KUKA KRL program: MyProgram_044().src

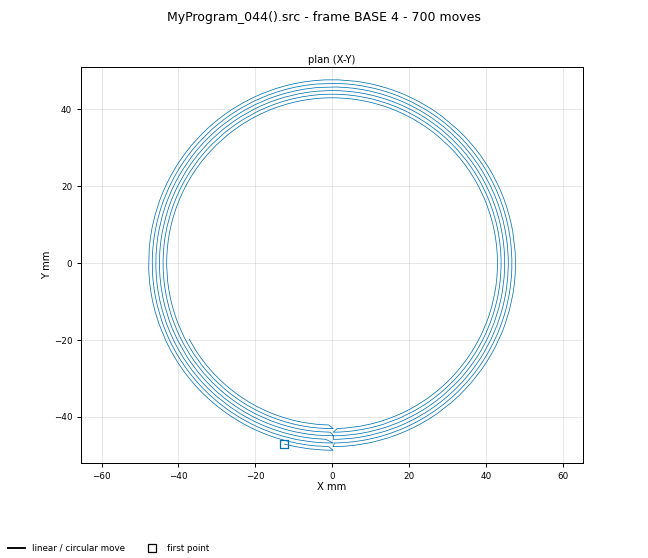
[picture p0: tool path of MyProgram_044().src in frame BASE 4, 700 of 700 moves have a stored position in this frame; points joined in program order, loops and branches not executed]
&ACCESS RVP
&REL 1
&PARAM TEMPLATE = C:\KRC\Roboter\Template\vorgabe
&PARAM EDITMASK = *
DEF MyProgram_044()
; ---- Setting reference (Base) ----
$BASE = BASE_DATA[4]

; --------------------------
; ---- Setting tool (TCP) ----
$TOOL = TOOL_DATA[3]
; --------------------------

$VEL.CP = VEL_APROX_PRINT
Startdeposition()
$VEL.CP = VEL_PRINT
LIN {X -12.395,Y -47.0783,Z 64,A -109.7384,B 24.8767,C -2.5626,E1 24.9625,E2 -526.6882} C_DIS
LIN {X -9.7511,Y -47.6962,Z 64,A -106.6183,B 24.877,C -2.56,E1 24.971,E2 -529.8057} C_DIS
LIN {X -6.2338,Y -48.282,Z 64,A -102.6118,B 24.8774,C -2.5558,E1 24.982,E2 -533.8056} C_DIS
LIN {X -2.3323,Y -48.6268,Z 64,A -98.0603,B 24.8774,C -2.5547,E1 24.9947,E2 -538.3566} C_DIS
LIN {X 0.2772,Y -48.6819,Z 64,A -96.4409,B 24.8798,C -2.5307,E1 24.9991,E2 -539.9189} C_DIS
Enddeposition()
LIN {X 0.2772,Y -48.6819,Z 64,A -96.4409,B 24.8798,C -2.5307,E1 24.9991,E2 -539.9189} C_DIS
Startdeposition()
$VEL.CP = VEL_PRINT
LIN {X -0.9286,Y -47.7351,Z 64,A -98.3994,B 24.879,C -2.5386,E1 24.9937,E2 -537.979} C_DIS
LIN {X -4.5581,Y -47.526,Z 64,A -101.7319,B 24.8774,C -2.5553,E1 24.9845,E2 -534.6849} C_DIS
LIN {X -6.6871,Y -47.2729,Z 64,A -104.8435,B 24.8782,C -2.5471,E1 24.9758,E2 -531.5515} C_DIS
LIN {X -9.333,Y -46.8231,Z 64,A -108.0485,B 24.8781,C -2.5484,E1 24.967,E2 -528.3464} C_DIS
LIN {X -12.0507,Y -46.1979,Z 64,A -111.4661,B 24.8781,C -2.549,E1 24.9577,E2 -524.9256} C_DIS
LIN {X -14.2576,Y -45.5655,Z 64,A -113.9601,B 24.8775,C -2.555,E1 24.9511,E2 -522.4415} C_DIS
LIN {X -16.0969,Y -44.9485,Z 64,A -116.3815,B 24.8775,C -2.5554,E1 24.9447,E2 -520.0165} C_DIS
LIN {X -17.8418,Y -44.2849,Z 64,A -118.4806,B 24.877,C -2.5597,E1 24.9392,E2 -517.923} C_DIS
LIN {X -19.622,Y -43.5255,Z 64,A -120.9789,B 24.877,C -2.5595,E1 24.9328,E2 -515.4183} C_DIS
LIN {X -21.7184,Y -42.5182,Z 64,A -123.9566,B 24.877,C -2.56,E1 24.9254,E2 -512.434} C_DIS
LIN {X -23.6622,Y -41.4683,Z 64,A -126.3379,B 24.8762,C -2.5675,E1 24.9196,E2 -510.0637} C_DIS
LIN {X -25.9488,Y -40.0766,Z 64,A -129.6657,B 24.8759,C -2.5705,E1 24.9117,E2 -506.7327} C_DIS
LIN {X -27.6681,Y -38.9099,Z 64,A -132.1587,B 24.8756,C -2.5746,E1 24.906,E2 -504.2408} C_DIS
LIN {X -29.7267,Y -37.361,Z 64,A -134.9829,B 24.8747,C -2.5838,E1 24.8997,E2 -501.4283} C_DIS
LIN {X -31.3956,Y -35.9696,Z 64,A -138.059,B 24.8748,C -2.5819,E1 24.8932,E2 -498.336} C_DIS
LIN {X -33.6241,Y -33.8958,Z 64,A -141.6218,B 24.874,C -2.5906,E1 24.886,E2 -494.779} C_DIS
LIN {X -35.3679,Y -32.073,Z 64,A -144.7793,B 24.8735,C -2.5952,E1 24.88,E2 -491.6188} C_DIS
LIN {X -37.2668,Y -29.8454,Z 64,A -148.2463,B 24.8727,C -2.6038,E1 24.8738,E2 -488.1564} C_DIS
LIN {X -38.4195,Y -28.3455,Z 64,A -150.8413,B 24.8727,C -2.6048,E1 24.8694,E2 -485.5513} C_DIS
LIN {X -40.21,Y -25.7421,Z 64,A -154.4257,B 24.8714,C -2.6171,E1 24.8639,E2 -481.9782} C_DIS
LIN {X -41.9231,Y -22.8465,Z 64,A -158.8875,B 24.8709,C -2.622,E1 24.8578,E2 -477.5049} C_DIS
LIN {X -43.2781,Y -20.1618,Z 64,A -162.6851,B 24.8702,C -2.6295,E1 24.8532,E2 -473.7045} C_DIS
LIN {X -45.1395,Y -15.5552,Z 64,A -168.6201,B 24.8684,C -2.6469,E1 24.8474,E2 -467.7776} C_DIS
LIN {X -46.1878,Y -12.0906,Z 64,A -172.3555,B 24.8664,C -2.6677,E1 24.8446,E2 -464.0703} C_DIS
LIN {X -46.7423,Y -9.73,Z 64,A -175.6447,B 24.866,C -2.6715,E1 24.8426,E2 -460.771} C_DIS
LIN {X -47.2314,Y -6.9813,Z 64,A -178.6079,B 24.8644,C -2.6868,E1 24.8413,E2 -457.8267} C_DIS
LIN {X -47.4828,Y -4.9862,Z 64,A 178.9355,B 24.8637,C -2.6937,E1 24.8405,E2 -455.3719} C_DIS
LIN {X -47.6696,Y -2.665,Z 64,A 176.3561,B 24.8626,C -2.7052,E1 24.84,E2 -452.8044} C_DIS
LIN {X -47.7273,Y -1.2631,Z 64,A 173.6261,B 24.8634,C -2.6971,E1 24.8398,E2 -450.0386} C_DIS
LIN {X -47.5831,Y 3.9179,Z 64,A 168.1994,B 24.8604,C -2.7268,E1 24.8405,E2 -444.6502} C_DIS
LIN {X -47.2564,Y 6.8067,Z 64,A 164.3377,B 24.8597,C -2.7329,E1 24.8418,E2 -440.7803} C_DIS
LIN {X -46.8079,Y 9.409,Z 64,A 161.4797,B 24.8583,C -2.7468,E1 24.8433,E2 -437.9385} C_DIS
LIN {X -46.0261,Y 12.6919,Z 64,A 156.8291,B 24.8578,C -2.7516,E1 24.8465,E2 -433.2723} C_DIS
LIN {X -44.8495,Y 16.3711,Z 64,A 153.1258,B 24.8551,C -2.7777,E1 24.8497,E2 -429.6103} C_DIS
LIN {X -44.1797,Y 18.1013,Z 64,A 150.357,B 24.8551,C -2.7773,E1 24.8526,E2 -426.8251} C_DIS
LIN {X -43.1295,Y 20.4774,Z 64,A 147.3798,B 24.854,C -2.7883,E1 24.8561,E2 -423.8579} C_DIS
LIN {X -42.0435,Y 22.6245,Z 64,A 143.9498,B 24.8538,C -2.7896,E1 24.8605,E2 -420.4125} C_DIS
LIN {X -40.5413,Y 25.2173,Z 64,A 140.8516,B 24.8521,C -2.8061,E1 24.8649,E2 -417.338} C_DIS
LIN {X -39.3814,Y 26.993,Z 64,A 138.1652,B 24.8515,C -2.8112,E1 24.8691,E2 -414.6502} C_DIS
LIN {X -38.0323,Y 28.8634,Z 64,A 135.3123,B 24.8509,C -2.8173,E1 24.8739,E2 -411.7984} C_DIS
LIN {X -36.3497,Y 30.9548,Z 64,A 132.0941,B 24.85,C -2.8256,E1 24.8796,E2 -408.5849} C_DIS
LIN {X -33.8073,Y 33.7137,Z 64,A 127.1095,B 24.8496,C -2.8299,E1 24.8892,E2 -403.5891} C_DIS
LIN {X -31.9372,Y 35.4898,Z 64,A 124.4061,B 24.8482,C -2.8422,E1 24.8947,E2 -400.9042} C_DIS
LIN {X -29.5152,Y 37.5281,Z 64,A 120.5281,B 24.8475,C -2.8493,E1 24.9031,E2 -397.0284} C_DIS
LIN {X -27.7313,Y 38.8648,Z 64,A 117.8178,B 24.847,C -2.8541,E1 24.9092,E2 -394.3202} C_DIS
LIN {X -25.7301,Y 40.2177,Z 64,A 114.9913,B 24.8463,C -2.8606,E1 24.9158,E2 -391.4999} C_DIS
LIN {X -22.9528,Y 41.8654,Z 64,A 111.0966,B 24.8456,C -2.867,E1 24.9253,E2 -387.609} C_DIS
LIN {X -20.5095,Y 43.1143,Z 64,A 107.8779,B 24.8449,C -2.8732,E1 24.9333,E2 -384.3968} C_DIS
LIN {X -18.1914,Y 44.1428,Z 64,A 104.6647,B 24.8447,C -2.8751,E1 24.9416,E2 -381.1804} C_DIS
LIN {X -14.6042,Y 45.4553,Z 64,A 99.8433,B 24.8445,C -2.8771,E1 24.9543,E2 -376.3547} C_DIS
LIN {X -11.9557,Y 46.2229,Z 64,A 97.1011,B 24.8432,C -2.8889,E1 24.9616,E2 -373.6364} C_DIS
LIN {X -9.839,Y 46.7195,Z 64,A 94.3332,B 24.8432,C -2.8889,E1 24.9692,E2 -370.8646} C_DIS
LIN {X -7.3492,Y 47.1751,Z 64,A 91.1356,B 24.8432,C -2.8885,E1 24.978,E2 -367.6633} C_DIS
LIN {X -4.4968,Y 47.5319,Z 64,A 88.0845,B 24.8424,C -2.8966,E1 24.9864,E2 -364.6294} C_DIS
LIN {X -1.7768,Y 47.7113,Z 64,A 84.2696,B 24.8431,C -2.8893,E1 24.9971,E2 -360.7961} C_DIS
LIN {X 1.6532,Y 47.7156,Z 64,A 79.8522,B 24.8436,C -2.8851,E1 25.0094,E2 -356.3695} C_DIS
LIN {X 5.8821,Y 47.3806,Z 64,A 75.7338,B 24.842,C -2.9002,E1 25.0208,E2 -352.2894} C_DIS
LIN {X 7.6244,Y 47.132,Z 64,A 72.7996,B 24.8435,C -2.8862,E1 25.029,E2 -349.3248} C_DIS
LIN {X 10.1643,Y 46.6496,Z 64,A 70.1964,B 24.8427,C -2.893,E1 25.036,E2 -346.741} C_DIS
LIN {X 12.1272,Y 46.178,Z 64,A 67.8281,B 24.8427,C -2.8925,E1 25.0424,E2 -344.3751} C_DIS
LIN {X 14.1267,Y 45.6062,Z 64,A 65.4726,B 24.8427,C -2.8931,E1 25.0487,E2 -342.025} C_DIS
LIN {X 15.6089,Y 45.1209,Z 64,A 63.3651,B 24.8433,C -2.8876,E1 25.0543,E2 -339.9085} C_DIS
LIN {X 17.816,Y 44.2953,Z 64,A 60.7762,B 24.8432,C -2.889,E1 25.061,E2 -337.3286} C_DIS
LIN {X 19.3175,Y 43.6614,Z 64,A 58.381,B 24.8442,C -2.8794,E1 25.0672,E2 -334.9163} C_DIS
LIN {X 21.7553,Y 42.4995,Z 64,A 55.2848,B 24.8444,C -2.8779,E1 25.075,E2 -331.8251} C_DIS
LIN {X 24.4911,Y 40.9843,Z 64,A 51.7991,B 24.8444,C -2.8774,E1 25.0834,E2 -328.3485} C_DIS
LIN {X 26.3871,Y 39.7898,Z 64,A 48.834,B 24.8454,C -2.8684,E1 25.0904,E2 -325.3718} C_DIS
LIN {X 28.4987,Y 38.3058,Z 64,A 45.1897,B 24.847,C -2.8536,E1 25.0986,E2 -321.7051} C_DIS
LIN {X 32.9673,Y 34.5352,Z 64,A 38.7549,B 24.8473,C -2.8505,E1 25.1121,E2 -315.2885} C_DIS
LIN {X 34.8438,Y 32.6407,Z 64,A 35.5678,B 24.848,C -2.844,E1 25.1183,E2 -312.0996} C_DIS
LIN {X 37.3566,Y 29.7323,Z 64,A 31.3931,B 24.8483,C -2.8416,E1 25.1258,E2 -307.9382} C_DIS
LIN {X 38.7827,Y 27.8463,Z 64,A 27.8779,B 24.8504,C -2.8222,E1 25.1317,E2 -304.3942} C_DIS
LIN {X 40.8107,Y 24.7787,Z 64,A 23.5188,B 24.8515,C -2.812,E1 25.1382,E2 -300.0329} C_DIS
LIN {X 42.0195,Y 22.6688,Z 64,A 20.888,B 24.8517,C -2.8096,E1 25.1417,E2 -297.4101} C_DIS
LIN {X 43.5018,Y 19.6746,Z 64,A 17.248,B 24.8521,C -2.8056,E1 25.1461,E2 -293.7802} C_DIS
LIN {X 44.5986,Y 17.0433,Z 64,A 13.8143,B 24.8532,C -2.7957,E1 25.1497,E2 -290.342} C_DIS
LIN {X 45.4386,Y 14.657,Z 64,A 10.0859,B 24.8555,C -2.7737,E1 25.1531,E2 -286.5826} C_DIS
LIN {X 46.4419,Y 11.0739,Z 64,A 6.0353,B 24.8561,C -2.7683,E1 25.1559,E2 -282.5425} C_DIS
LIN {X 47.015,Y 8.3123,Z 64,A 1.8245,B 24.8588,C -2.7422,E1 25.1581,E2 -278.2946} C_DIS
LIN {X 47.6603,Y 2.8333,Z 64,A -3.3532,B 24.858,C -2.7494,E1 25.1595,E2 -273.1646} C_DIS
LIN {X 47.7412,Y -0.5621,Z 64,A -7.8342,B 24.8602,C -2.7287,E1 25.1597,E2 -268.6614} C_DIS
LIN {X 47.6513,Y -2.9787,Z 64,A -10.826,B 24.8613,C -2.7179,E1 25.1593,E2 -265.6617} C_DIS
LIN {X 47.4135,Y -5.6084,Z 64,A -14.0861,B 24.8625,C -2.7061,E1 25.1584,E2 -262.3931} C_DIS
LIN {X 47.0566,Y -8.0754,Z 64,A -17.2852,B 24.8638,C -2.6928,E1 25.1569,E2 -259.1812} C_DIS
LIN {X 46.1862,Y -12.0964,Z 64,A -22.4469,B 24.8658,C -2.6731,E1 25.1535,E2 -254.003} C_DIS
LIN {X 44.9125,Y -16.1976,Z 64,A -26.7244,B 24.8658,C -2.6742,E1 25.1498,E2 -249.7522} C_DIS
LIN {X 44.2181,Y -18.0066,Z 64,A -29.8233,B 24.8679,C -2.6524,E1 25.1466,E2 -246.6189} C_DIS
LIN {X 42.6286,Y -21.5011,Z 64,A -33.8951,B 24.8682,C -2.6491,E1 25.1417,E2 -242.5612} C_DIS
LIN {X 41.547,Y -23.5236,Z 64,A -36.6489,B 24.869,C -2.6412,E1 25.1379,E2 -239.8031} C_DIS
LIN {X 39.9965,Y -26.0726,Z 64,A -39.9883,B 24.8695,C -2.6359,E1 25.133,E2 -236.4678} C_DIS
LIN {X 38.9178,Y -27.657,Z 64,A -42.8338,B 24.8712,C -2.6194,E1 25.1284,E2 -233.5972} C_DIS
LIN {X 36.2013,Y -31.1289,Z 64,A -48.2812,B 24.8728,C -2.6028,E1 25.1187,E2 -228.1358} C_DIS
LIN {X 33.0813,Y -34.4257,Z 64,A -52.6432,B 24.8721,C -2.61,E1 25.1103,E2 -223.8094} C_DIS
LIN {X 31.1165,Y -36.2119,Z 64,A -56.8723,B 24.8747,C -2.5835,E1 25.1013,E2 -219.5346} C_DIS
LIN {X 27.4183,Y -39.0865,Z 64,A -62.2626,B 24.8754,C -2.5762,E1 25.0893,E2 -214.1462} C_DIS
LIN {X 24.9285,Y -40.7196,Z 64,A -65.4708,B 24.8754,C -2.5762,E1 25.0817,E2 -210.9481} C_DIS
LIN {X 22.8449,Y -41.9239,Z 64,A -68.1053,B 24.8754,C -2.5757,E1 25.0753,E2 -208.3202} C_DIS
LIN {X 21.2981,Y -42.7305,Z 64,A -70.0628,B 24.8755,C -2.5747,E1 25.0705,E2 -206.3658} C_DIS
LIN {X 19.467,Y -43.5948,Z 64,A -72.895,B 24.8766,C -2.5638,E1 25.0632,E2 -203.515} C_DIS
LIN {X 16.541,Y -44.7873,Z 64,A -76.6485,B 24.877,C -2.5594,E1 25.0534,E2 -199.7592} C_DIS
LIN {X 14.4167,Y -45.5152,Z 64,A -79.4404,B 24.8775,C -2.5545,E1 25.046,E2 -196.9609} C_DIS
LIN {X 11.2342,Y -46.4033,Z 64,A -83.1494,B 24.8775,C -2.5548,E1 25.036,E2 -193.2586} C_DIS
LIN {X 9.527,Y -46.7839,Z 64,A -85.5211,B 24.8781,C -2.5484,E1 25.0295,E2 -190.8745} C_DIS
LIN {X 5.9203,Y -47.376,Z 64,A -89.4382,B 24.8776,C -2.5533,E1 25.0187,E2 -186.9727} C_DIS
LIN {X 3.4815,Y -47.6175,Z 64,A -92.9139,B 24.8786,C -2.5429,E1 25.009,E2 -183.4742} C_DIS
LIN {X 0.2827,Y -47.7422,Z 64,A -96.3741,B 24.8781,C -2.548,E1 24.9994,E2 -180.0269} C_DIS
Enddeposition()
LIN {X 0.2827,Y -47.7422,Z 64,A -96.3741,B 24.8781,C -2.548,E1 24.9994,E2 -180.0269} C_DIS
Startdeposition()
$VEL.CP = VEL_PRINT
LIN {X 0.6342,Y -46.8012,Z 64,A -94.7946,B 24.8747,C -2.5833,E1 25.004,E2 -181.6901} C_DIS
LIN {X 3.085,Y -46.7035,Z 64,A -91.5094,B 24.8741,C -2.5892,E1 25.0132,E2 -184.9881} C_DIS
LIN {X 5.746,Y -46.4516,Z 64,A -88.1759,B 24.8739,C -2.5921,E1 25.0225,E2 -188.3263} C_DIS
LIN {X 8.6832,Y -45.9928,Z 64,A -84.6953,B 24.8739,C -2.5921,E1 25.032,E2 -191.8032} C_DIS
LIN {X 11.2628,Y -45.4303,Z 64,A -81.3653,B 24.8734,C -2.5969,E1 25.0411,E2 -195.1398} C_DIS
LIN {X 13.3341,Y -44.8658,Z 64,A -79.1038,B 24.8737,C -2.5933,E1 25.0472,E2 -197.3892} C_DIS
LIN {X 15.2084,Y -44.2657,Z 64,A -76.2089,B 24.8726,C -2.6048,E1 25.0549,E2 -200.3056} C_DIS
LIN {X 17.9227,Y -43.2382,Z 64,A -72.9255,B 24.8726,C -2.6048,E1 25.0634,E2 -203.5819} C_DIS
LIN {X 19.8547,Y -42.3857,Z 64,A -70.4518,B 24.8724,C -2.6068,E1 25.0697,E2 -206.054} C_DIS
LIN {X 21.779,Y -41.4296,Z 64,A -68.1334,B 24.8725,C -2.6055,E1 25.0754,E2 -208.3629} C_DIS
LIN {X 23.3037,Y -40.5916,Z 64,A -65.6769,B 24.8716,C -2.6151,E1 25.0814,E2 -210.8349} C_DIS
LIN {X 24.9354,Y -39.6105,Z 64,A -63.532,B 24.8716,C -2.616,E1 25.0865,E2 -212.9752} C_DIS
LIN {X 27.0041,Y -38.2303,Z 64,A -59.9123,B 24.8699,C -2.6325,E1 25.0949,E2 -216.6217} C_DIS
LIN {X 29.2839,Y -36.5134,Z 64,A -56.5753,B 24.8694,C -2.637,E1 25.1023,E2 -219.9569} C_DIS
LIN {X 31.5484,Y -34.5753,Z 64,A -53.3242,B 24.8694,C -2.6378,E1 25.109,E2 -223.1971} C_DIS
LIN {X 32.9023,Y -33.2893,Z 64,A -50.715,B 24.8682,C -2.6492,E1 25.1143,E2 -225.8224} C_DIS
LIN {X 35.0123,Y -31.0632,Z 64,A -47.2319,B 24.8678,C -2.6534,E1 25.1209,E2 -229.3} C_DIS
LIN {X 36.8334,Y -28.8804,Z 64,A -43.3302,B 24.8661,C -2.6703,E1 25.1278,E2 -233.2238} C_DIS
LIN {X 38.3039,Y -26.8994,Z 64,A -40.9216,B 24.8665,C -2.6668,E1 25.1317,E2 -235.6124} C_DIS
LIN {X 39.2605,Y -25.4833,Z 64,A -38.6906,B 24.8656,C -2.6752,E1 25.1351,E2 -237.8521} C_DIS
LIN {X 40.4459,Y -23.5571,Z 64,A -35.7988,B 24.8646,C -2.6853,E1 25.1393,E2 -240.7531} C_DIS
LIN {X 41.8282,Y -21.0041,Z 64,A -32.3163,B 24.8637,C -2.6942,E1 25.1438,E2 -244.2382} C_DIS
LIN {X 43.0084,Y -18.4673,Z 64,A -28.7338,B 24.8623,C -2.7074,E1 25.1479,E2 -247.8323} C_DIS
LIN {X 43.9827,Y -16.0083,Z 64,A -25.6523,B 24.8617,C -2.7141,E1 25.1509,E2 -250.9126} C_DIS
LIN {X 44.7903,Y -13.5846,Z 64,A -22.3402,B 24.8603,C -2.7273,E1 25.1537,E2 -254.2371} C_DIS
LIN {X 45.413,Y -11.3318,Z 64,A -19.2917,B 24.859,C -2.7398,E1 25.1558,E2 -257.2976} C_DIS
LIN {X 46.0028,Y -8.6308,Z 64,A -16.6613,B 24.8594,C -2.7357,E1 25.1573,E2 -259.903} C_DIS
LIN {X 46.339,Y -6.59,Z 64,A -13.4915,B 24.8573,C -2.756,E1 25.1586,E2 -263.1023} C_DIS
LIN {X 46.6589,Y -3.7003,Z 64,A -10.2295,B 24.8568,C -2.7615,E1 25.1595,E2 -266.3577} C_DIS
LIN {X 46.7751,Y -1.6919,Z 64,A -7.9435,B 24.8563,C -2.7658,E1 25.1597,E2 -268.6403} C_DIS
LIN {X 46.7921,Y 1.1,Z 64,A -4.3105,B 24.8548,C -2.7807,E1 25.1597,E2 -272.2869} C_DIS
LIN {X 46.6119,Y 4.247,Z 64,A -0.573,B 24.8537,C -2.7904,E1 25.1589,E2 -276.0252} C_DIS
LIN {X 46.3482,Y 6.5248,Z 64,A 2.0753,B 24.8532,C -2.796,E1 25.1579,E2 -278.6711} C_DIS
LIN {X 46.0174,Y 8.5543,Z 64,A 4.5784,B 24.8524,C -2.8034,E1 25.1567,E2 -281.1771} C_DIS
LIN {X 45.5613,Y 10.7204,Z 64,A 7.2402,B 24.8516,C -2.8106,E1 25.1551,E2 -283.8406} C_DIS
LIN {X 45.1148,Y 12.4653,Z 64,A 9.2143,B 24.8514,C -2.8128,E1 25.1537,E2 -285.8085} C_DIS
LIN {X 44.5439,Y 14.3732,Z 64,A 11.9778,B 24.8499,C -2.8262,E1 25.1514,E2 -288.588} C_DIS
LIN {X 43.6644,Y 16.8579,Z 64,A 15.1569,B 24.8491,C -2.8345,E1 25.1483,E2 -291.769} C_DIS
LIN {X 42.7002,Y 19.1685,Z 64,A 18.2894,B 24.848,C -2.8444,E1 25.1448,E2 -294.9077} C_DIS
LIN {X 41.3826,Y 21.8684,Z 64,A 21.5209,B 24.8478,C -2.846,E1 25.1408,E2 -298.1258} C_DIS
LIN {X 40.1234,Y 24.102,Z 64,A 25.3236,B 24.8456,C -2.8666,E1 25.1354,E2 -301.9577} C_DIS
LIN {X 38.9075,Y 26.0191,Z 64,A 27.9514,B 24.8452,C -2.8708,E1 25.1314,E2 -304.5823} C_DIS
LIN {X 37.0697,Y 28.5758,Z 64,A 31.3241,B 24.8452,C -2.8711,E1 25.1258,E2 -307.9396} C_DIS
LIN {X 34.9763,Y 31.1035,Z 64,A 35.5365,B 24.8438,C -2.8837,E1 25.1182,E2 -312.1627} C_DIS
LIN {X 33.2605,Y 32.9315,Z 64,A 38.6668,B 24.8429,C -2.8914,E1 25.1121,E2 -315.2976} C_DIS
LIN {X 30.5308,Y 35.4771,Z 64,A 43.0808,B 24.8422,C -2.8975,E1 25.103,E2 -319.7084} C_DIS
LIN {X 28.9107,Y 36.8094,Z 64,A 45.5609,B 24.8419,C -2.9006,E1 25.0976,E2 -322.1865} C_DIS
LIN {X 27.5077,Y 37.8695,Z 64,A 47.646,B 24.8416,C -2.9031,E1 25.0929,E2 -324.2699} C_DIS
LIN {X 25.2892,Y 39.3853,Z 64,A 51.0253,B 24.8409,C -2.9099,E1 25.085,E2 -327.6541} C_DIS
LIN {X 23.7995,Y 40.3029,Z 64,A 53.5315,B 24.8399,C -2.9193,E1 25.079,E2 -330.175} C_DIS
LIN {X 20.5147,Y 42.0701,Z 64,A 58.282,B 24.8389,C -2.9283,E1 25.0672,E2 -334.9336} C_DIS
LIN {X 17.0842,Y 43.5761,Z 64,A 62.1836,B 24.8396,C -2.9213,E1 25.0572,E2 -338.8095} C_DIS
LIN {X 15.4042,Y 44.198,Z 64,A 64.4907,B 24.8392,C -2.9251,E1 25.0511,E2 -341.121} C_DIS
LIN {X 13.3641,Y 44.8567,Z 64,A 67.1244,B 24.839,C -2.9272,E1 25.0441,E2 -343.755} C_DIS
LIN {X 10.9256,Y 45.5122,Z 64,A 70.2327,B 24.8388,C -2.9293,E1 25.0357,E2 -346.8635} C_DIS
LIN {X 7.819,Y 46.1476,Z 64,A 73.9653,B 24.8388,C -2.9285,E1 25.0255,E2 -350.5896} C_DIS
LIN {X 5.9098,Y 46.4308,Z 64,A 76.3697,B 24.8388,C -2.9297,E1 25.0188,E2 -352.9949} C_DIS
LIN {X 3.7771,Y 46.6527,Z 64,A 79.2175,B 24.8383,C -2.9335,E1 25.0109,E2 -355.8502} C_DIS
LIN {X 1.1995,Y 46.7899,Z 64,A 83.0787,B 24.8371,C -2.9445,E1 25,E2 -359.7366} C_DIS
LIN {X -3.9742,Y 46.6363,Z 64,A 88.5906,B 24.8388,C -2.9292,E1 24.9848,E2 -365.2136} C_DIS
LIN {X -6.8684,Y 46.2987,Z 64,A 92.4777,B 24.8385,C -2.932,E1 24.974,E2 -369.1102} C_DIS
LIN {X -9.36,Y 45.8599,Z 64,A 95.1805,B 24.8394,C -2.9236,E1 24.9666,E2 -371.7959} C_DIS
LIN {X -11.4862,Y 45.3743,Z 64,A 97.9922,B 24.8394,C -2.9233,E1 24.959,E2 -374.6107} C_DIS
LIN {X -14.1559,Y 44.6132,Z 64,A 101.7915,B 24.8392,C -2.9256,E1 24.9488,E2 -378.4219} C_DIS
LIN {X -16.5969,Y 43.764,Z 64,A 105.3784,B 24.8389,C -2.9278,E1 24.9394,E2 -382.0215} C_DIS
LIN {X -20.1209,Y 42.2596,Z 64,A 109.38,B 24.8408,C -2.9108,E1 24.9293,E2 -385.9923} C_DIS
LIN {X -23.5707,Y 40.4364,Z 64,A 114.4699,B 24.8412,C -2.9073,E1 24.9168,E2 -391.0884} C_DIS
LIN {X -25.9496,Y 38.9535,Z 64,A 117.5019,B 24.8425,C -2.8952,E1 24.9097,E2 -394.1014} C_DIS
LIN {X -27.9755,Y 37.5252,Z 64,A 120.6772,B 24.8429,C -2.8911,E1 24.9026,E2 -397.278} C_DIS
LIN {X -30.2011,Y 35.7586,Z 64,A 124.1179,B 24.8438,C -2.8832,E1 24.8951,E2 -400.7127} C_DIS
LIN {X -31.6166,Y 34.5128,Z 64,A 126.9902,B 24.8435,C -2.8857,E1 24.8892,E2 -403.6028} C_DIS
LIN {X -34.6929,Y 31.4191,Z 64,A 131.8617,B 24.8456,C -2.8665,E1 24.8798,E2 -408.4493} C_DIS
LIN {X -36.4484,Y 29.3645,Z 64,A 135.1345,B 24.8466,C -2.8576,E1 24.874,E2 -411.7159} C_DIS
LIN {X -37.6336,Y 27.8299,Z 64,A 137.8335,B 24.8468,C -2.8557,E1 24.8695,E2 -414.4234} C_DIS
LIN {X -39.4095,Y 25.2514,Z 64,A 141.4179,B 24.8483,C -2.842,E1 24.864,E2 -417.9929} C_DIS
LIN {X -41.0331,Y 22.5172,Z 64,A 145.9162,B 24.8486,C -2.839,E1 24.8577,E2 -422.5076} C_DIS
LIN {X -42.3743,Y 19.8791,Z 64,A 149.375,B 24.8499,C -2.8262,E1 24.8536,E2 -425.9547} C_DIS
LIN {X -43.7887,Y 16.5316,Z 64,A 153.3349,B 24.852,C -2.8066,E1 24.8495,E2 -429.8896} C_DIS
LIN {X -44.6099,Y 14.1663,Z 64,A 156.814,B 24.8524,C -2.8027,E1 24.8464,E2 -433.3792} C_DIS
LIN {X -45.5232,Y 10.8797,Z 64,A 160.7905,B 24.8541,C -2.7872,E1 24.8436,E2 -437.3419} C_DIS
LIN {X -46.0725,Y 8.2504,Z 64,A 163.9661,B 24.8553,C -2.7755,E1 24.842,E2 -440.5082} C_DIS
LIN {X -46.4192,Y 5.9983,Z 64,A 166.8986,B 24.856,C -2.7686,E1 24.8408,E2 -443.4418} C_DIS
LIN {X -46.6752,Y 3.4923,Z 64,A 169.4985,B 24.8577,C -2.7527,E1 24.8402,E2 -446.0192} C_DIS
LIN {X -46.7964,Y 0.9112,Z 64,A 173.5745,B 24.8575,C -2.7545,E1 24.8398,E2 -450.1241} C_DIS
LIN {X -46.7535,Y -2.1957,Z 64,A 176.9979,B 24.8592,C -2.7377,E1 24.8401,E2 -453.5279} C_DIS
LIN {X -46.6217,Y -4.1413,Z 64,A 179.4719,B 24.8599,C -2.7314,E1 24.8407,E2 -456.0016} C_DIS
LIN {X -46.3019,Y -6.85,Z 64,A -177.6073,B 24.8615,C -2.7157,E1 24.8417,E2 -458.9023} C_DIS
LIN {X -46.0802,Y -8.2066,Z 64,A -175.3508,B 24.8613,C -2.718,E1 24.8428,E2 -461.1778} C_DIS
LIN {X -45.4603,Y -11.1404,Z 64,A -171.8246,B 24.8626,C -2.705,E1 24.845,E2 -464.6937} C_DIS
LIN {X -44.2097,Y -15.3707,Z 64,A -166.0866,B 24.8637,C -2.6937,E1 24.8498,E2 -470.4374} C_DIS
LIN {X -43.0201,Y -18.4394,Z 64,A -162.6722,B 24.8657,C -2.6741,E1 24.8533,E2 -473.8241} C_DIS
LIN {X -42.3744,Y -19.8785,Z 64,A -160.6968,B 24.8662,C -2.6694,E1 24.8556,E2 -475.799} C_DIS
LIN {X -41.701,Y -21.2545,Z 64,A -158.4981,B 24.8662,C -2.6686,E1 24.8584,E2 -478.0078} C_DIS
LIN {X -40.4073,Y -23.6221,Z 64,A -155.4706,B 24.8675,C -2.6562,E1 24.8625,E2 -481.0215} C_DIS
LIN {X -39.1654,Y -25.6288,Z 64,A -152.5662,B 24.8682,C -2.6491,E1 24.8669,E2 -483.9237} C_DIS
LIN {X -37.4149,Y -28.1223,Z 64,A -148.5392,B 24.8687,C -2.6442,E1 24.8734,E2 -487.9584} C_DIS
LIN {X -35.6448,Y -30.3346,Z 64,A -144.7853,B 24.8691,C -2.6402,E1 24.8801,E2 -491.7203} C_DIS
LIN {X -33.9869,Y -32.1817,Z 64,A -141.5829,B 24.8695,C -2.636,E1 24.8863,E2 -494.9267} C_DIS
LIN {X -31.8502,Y -34.2976,Z 64,A -138.2021,B 24.8707,C -2.6244,E1 24.8931,E2 -498.2936} C_DIS
LIN {X -29.4531,Y -36.3766,Z 64,A -134.8763,B 24.8722,C -2.6092,E1 24.9001,E2 -501.596} C_DIS
LIN {X -27.4013,Y -37.9465,Z 64,A -131.5451,B 24.8725,C -2.6062,E1 24.9075,E2 -504.932} C_DIS
LIN {X -26.2155,Y -38.7749,Z 64,A -129.4028,B 24.8722,C -2.6088,E1 24.9125,E2 -507.0877} C_DIS
LIN {X -23.7348,Y -40.3412,Z 64,A -125.8842,B 24.8728,C -2.6025,E1 24.9209,E2 -510.6023} C_DIS
LIN {X -21.2142,Y -41.7215,Z 64,A -122.2182,B 24.8731,C -2.6003,E1 24.9299,E2 -514.2731} C_DIS
LIN {X -19.144,Y -42.7112,Z 64,A -119.7825,B 24.8739,C -2.5915,E1 24.9361,E2 -516.694} C_DIS
LIN {X -17.3939,Y -43.4531,Z 64,A -117.2986,B 24.8739,C -2.5916,E1 24.9425,E2 -519.1837} C_DIS
LIN {X -15.3149,Y -44.2293,Z 64,A -114.1502,B 24.8735,C -2.596,E1 24.9508,E2 -522.3487} C_DIS
LIN {X -12.8555,Y -45.0054,Z 64,A -110.7564,B 24.8733,C -2.5976,E1 24.96,E2 -525.752} C_DIS
LIN {X -9.964,Y -45.7325,Z 64,A -107.9206,B 24.8747,C -2.5829,E1 24.9676,E2 -528.5566} C_DIS
LIN {X -8.5188,Y -46.0242,Z 64,A -105.5194,B 24.8739,C -2.5918,E1 24.9742,E2 -530.9814} C_DIS
LIN {X -4.7848,Y -46.56,Z 64,A -101.1924,B 24.8744,C -2.5863,E1 24.9862,E2 -535.2985} C_DIS
LIN {X -2.7262,Y -46.7258,Z 64,A -98.6042,B 24.8744,C -2.5874,E1 24.9934,E2 -537.89} C_DIS
LIN {X 0.2899,Y -46.7986,Z 64,A -96.5083,B 24.8768,C -2.5621,E1 24.9991,E2 -539.9261} C_DIS
Enddeposition()
LIN {X 0.2899,Y -46.7986,Z 64,A -96.5083,B 24.8768,C -2.5621,E1 24.9991,E2 -539.9261} C_DIS
Startdeposition()
$VEL.CP = VEL_PRINT
LIN {X -1.6444,Y -45.8371,Z 64,A -99.7182,B 24.8764,C -2.5659,E1 24.9902,E2 -536.7246} C_DIS
LIN {X -4.8851,Y -45.6056,Z 64,A -102.718,B 24.8748,C -2.5824,E1 24.9819,E2 -533.7626} C_DIS
LIN {X -6.7079,Y -45.3739,Z 64,A -105.1635,B 24.875,C -2.5805,E1 24.9751,E2 -531.3108} C_DIS
LIN {X -8.719,Y -45.0303,Z 64,A -107.7698,B 24.875,C -2.5805,E1 24.968,E2 -528.7018} C_DIS
LIN {X -10.9386,Y -44.5432,Z 64,A -110.5241,B 24.8747,C -2.5831,E1 24.9605,E2 -525.9501} C_DIS
LIN {X -12.6995,Y -44.0734,Z 64,A -113.0005,B 24.8749,C -2.5816,E1 24.9538,E2 -523.4662} C_DIS
LIN {X -15.3679,Y -43.2154,Z 64,A -116.7534,B 24.8749,C -2.5807,E1 24.9439,E2 -519.7041} C_DIS
LIN {X -18.1645,Y -42.1169,Z 64,A -120.156,B 24.8741,C -2.5895,E1 24.9351,E2 -516.3147} C_DIS
LIN {X -20.1395,Y -41.2086,Z 64,A -122.8725,B 24.8738,C -2.5925,E1 24.9282,E2 -513.5986} C_DIS
LIN {X -22.472,Y -39.9847,Z 64,A -125.8961,B 24.873,C -2.6006,E1 24.9208,E2 -510.5857} C_DIS
LIN {X -23.9885,Y -39.0937,Z 64,A -128.8256,B 24.8737,C -2.5935,E1 24.9138,E2 -507.6302} C_DIS
LIN {X -26.2953,Y -37.5804,Z 64,A -132.7571,B 24.8738,C -2.5923,E1 24.9047,E2 -503.6827} C_DIS
LIN {X -29.8183,Y -34.8515,Z 64,A -137.3802,B 24.8716,C -2.6151,E1 24.8947,E2 -499.0966} C_DIS
LIN {X -31.8833,Y -32.9728,Z 64,A -140.9945,B 24.8711,C -2.6203,E1 24.8874,E2 -495.48} C_DIS
LIN {X -33.6222,Y -31.1985,Z 64,A -143.9678,B 24.8703,C -2.6286,E1 24.8816,E2 -492.5136} C_DIS
LIN {X -34.6856,Y -30.0115,Z 64,A -146.5806,B 24.8706,C -2.6248,E1 24.8768,E2 -489.88} C_DIS
LIN {X -36.5496,Y -27.7114,Z 64,A -150.6684,B 24.8703,C -2.6285,E1 24.8698,E2 -485.7815} C_DIS
LIN {X -38.5002,Y -24.9302,Z 64,A -154.9483,B 24.8693,C -2.6387,E1 24.8632,E2 -481.5045} C_DIS
LIN {X -40.1793,Y -22.1229,Z 64,A -157.9202,B 24.8668,C -2.6634,E1 24.8592,E2 -478.5763} C_DIS
LIN {X -41.1239,Y -20.3117,Z 64,A -160.8046,B 24.8665,C -2.6661,E1 24.8555,E2 -475.6829} C_DIS
LIN {X -42.2059,Y -17.956,Z 64,A -164.2136,B 24.8658,C -2.673,E1 24.8516,E2 -472.2715} C_DIS
LIN {X -43.2718,Y -15.2087,Z 64,A -168.0594,B 24.865,C -2.6815,E1 24.8479,E2 -468.4244} C_DIS
LIN {X -44.301,Y -11.8818,Z 64,A -171.9257,B 24.8631,C -2.7003,E1 24.8449,E2 -464.5807} C_DIS
LIN {X -44.8135,Y -9.7725,Z 64,A -174.9708,B 24.8627,C -2.7044,E1 24.843,E2 -461.5274} C_DIS
LIN {X -45.2438,Y -7.533,Z 64,A -177.4649,B 24.8613,C -2.7174,E1 24.8418,E2 -459.0498} C_DIS
LIN {X -45.5066,Y -5.7371,Z 64,A -179.9593,B 24.8609,C -2.7216,E1 24.8408,E2 -456.5505} C_DIS
LIN {X -45.7487,Y -3.2846,Z 64,A 176.8311,B 24.8601,C -2.7296,E1 24.84,E2 -453.3407} C_DIS
LIN {X -45.8575,Y -0.9171,Z 64,A 173.6759,B 24.8594,C -2.7365,E1 24.8398,E2 -450.1829} C_DIS
LIN {X -45.8059,Y 2.3515,Z 64,A 169.7422,B 24.8578,C -2.7511,E1 24.8401,E2 -446.2606} C_DIS
LIN {X -45.6107,Y 4.8396,Z 64,A 166.6976,B 24.8567,C -2.7618,E1 24.8409,E2 -443.2232} C_DIS
LIN {X -45.3173,Y 7.0778,Z 64,A 163.9254,B 24.8558,C -2.7712,E1 24.842,E2 -440.4571} C_DIS
LIN {X -45.047,Y 8.6319,Z 64,A 161.476,B 24.8558,C -2.7715,E1 24.8433,E2 -437.994} C_DIS
LIN {X -44.2224,Y 12.1705,Z 64,A 157.0419,B 24.8541,C -2.7868,E1 24.8463,E2 -433.5706} C_DIS
LIN {X -43.4522,Y 14.6849,Z 64,A 154.1452,B 24.8526,C -2.8016,E1 24.8487,E2 -430.6926} C_DIS
LIN {X -42.8802,Y 16.28,Z 64,A 151.7301,B 24.8523,C -2.8043,E1 24.8511,E2 -428.2704} C_DIS
LIN {X -41.8108,Y 18.8572,Z 64,A 148.2049,B 24.8512,C -2.8141,E1 24.855,E2 -424.7492} C_DIS
LIN {X -40.7314,Y 21.0881,Z 64,A 145.3361,B 24.85,C -2.8259,E1 24.8585,E2 -421.8931} C_DIS
LIN {X -39.766,Y 22.8564,Z 64,A 142.6406,B 24.8495,C -2.8308,E1 24.8622,E2 -419.1952} C_DIS
LIN {X -38.8342,Y 24.4063,Z 64,A 139.9723,B 24.8493,C -2.832,E1 24.8662,E2 -416.5161} C_DIS
LIN {X -36.6076,Y 27.6342,Z 64,A 135.6592,B 24.8471,C -2.8524,E1 24.8731,E2 -412.2307} C_DIS
LIN {X -35.2612,Y 29.3325,Z 64,A 132.5107,B 24.8471,C -2.8537,E1 24.8787,E2 -409.0707} C_DIS
LIN {X -33.5949,Y 31.2278,Z 64,A 129.363,B 24.8462,C -2.8615,E1 24.8846,E2 -405.9276} C_DIS
LIN {X -31.486,Y 33.3525,Z 64,A 125.9701,B 24.8447,C -2.8747,E1 24.8913,E2 -402.5521} C_DIS
LIN {X -29.948,Y 34.7405,Z 64,A 123.6132,B 24.8438,C -2.8835,E1 24.8962,E2 -400.2068} C_DIS
LIN {X -28.5423,Y 35.9041,Z 64,A 120.9883,B 24.8438,C -2.8838,E1 24.9019,E2 -397.5728} C_DIS
LIN {X -25.5389,Y 38.0989,Z 64,A 116.302,B 24.8428,C -2.8925,E1 24.9126,E2 -392.8909} C_DIS
LIN {X -22.8772,Y 39.754,Z 64,A 111.7336,B 24.843,C -2.8907,E1 24.9235,E2 -388.3044} C_DIS
LIN {X -19.9461,Y 41.3026,Z 64,A 107.6538,B 24.8422,C -2.898,E1 24.9337,E2 -384.2313} C_DIS
LIN {X -16.4279,Y 42.8239,Z 64,A 103.6415,B 24.8403,C -2.9154,E1 24.944,E2 -380.2513} C_DIS
LIN {X -15.1283,Y 43.2998,Z 64,A 101.428,B 24.8408,C -2.9107,E1 24.9498,E2 -378.0223} C_DIS
LIN {X -12.4332,Y 44.1494,Z 64,A 97.9036,B 24.8404,C -2.9146,E1 24.9593,E2 -374.5012} C_DIS
LIN {X -9.4352,Y 44.8855,Z 64,A 94.2735,B 24.8396,C -2.9213,E1 24.9691,E2 -370.8823} C_DIS
LIN {X -7.2288,Y 45.294,Z 64,A 91.431,B 24.8395,C -2.9228,E1 24.9769,E2 -368.0405} C_DIS
LIN {X -4.7444,Y 45.6206,Z 64,A 88.5263,B 24.8389,C -2.9279,E1 24.985,E2 -365.146} C_DIS
LIN {X -3.2274,Y 45.7526,Z 64,A 85.7364,B 24.8403,C -2.9155,E1 24.9928,E2 -362.3257} C_DIS
LIN {X 1.0048,Y 45.8558,Z 64,A 81.1245,B 24.839,C -2.9268,E1 25.0056,E2 -357.7406} C_DIS
LIN {X 3.3168,Y 45.747,Z 64,A 78.3493,B 24.8388,C -2.9286,E1 25.0133,E2 -354.9707} C_DIS
LIN {X 5.485,Y 45.5376,Z 64,A 75.4286,B 24.8392,C -2.9251,E1 25.0215,E2 -352.0438} C_DIS
LIN {X 8.0141,Y 45.1611,Z 64,A 72.4582,B 24.8389,C -2.9277,E1 25.0296,E2 -349.0823} C_DIS
LIN {X 9.6602,Y 44.838,Z 64,A 70.0781,B 24.8395,C -2.9222,E1 25.0362,E2 -346.6923} C_DIS
LIN {X 12.4449,Y 44.1461,Z 64,A 66.3288,B 24.8401,C -2.9174,E1 25.0463,E2 -342.9374} C_DIS
LIN {X 15.1996,Y 43.275,Z 64,A 62.9616,B 24.84,C -2.9184,E1 25.0552,E2 -339.579} C_DIS
LIN {X 17.5757,Y 42.3659,Z 64,A 59.7085,B 24.8404,C -2.9141,E1 25.0636,E2 -336.3229} C_DIS
LIN {X 19.8447,Y 41.3514,Z 64,A 56.7665,B 24.8405,C -2.9132,E1 25.0711,E2 -333.3864} C_DIS
LIN {X 21.9899,Y 40.2518,Z 64,A 53.6678,B 24.8411,C -2.9079,E1 25.0787,E2 -330.2837} C_DIS
LIN {X 24.1788,Y 38.9762,Z 64,A 50.7667,B 24.8411,C -2.9077,E1 25.0857,E2 -327.3913} C_DIS
LIN {X 26.1545,Y 37.6788,Z 64,A 47.714,B 24.8418,C -2.9014,E1 25.0928,E2 -324.3337} C_DIS
LIN {X 27.8331,Y 36.4566,Z 64,A 45.2832,B 24.842,C -2.8997,E1 25.0982,E2 -321.9077} C_DIS
LIN {X 28.9991,Y 35.5363,Z 64,A 43.1912,B 24.8428,C -2.8923,E1 25.1028,E2 -319.8059} C_DIS
LIN {X 30.8372,Y 33.9534,Z 64,A 40.2316,B 24.8433,C -2.8877,E1 25.109,E2 -316.8471} C_DIS
LIN {X 32.5275,Y 32.3378,Z 64,A 36.5786,B 24.8454,C -2.8689,E1 25.1163,E2 -313.1651} C_DIS
LIN {X 34.5974,Y 30.1127,Z 64,A 33.1844,B 24.8455,C -2.8675,E1 25.1225,E2 -309.7828} C_DIS
LIN {X 36.3961,Y 27.912,Z 64,A 29.8786,B 24.8459,C -2.8636,E1 25.1283,E2 -306.4831} C_DIS
LIN {X 37.9853,Y 25.7074,Z 64,A 26.786,B 24.8463,C -2.8607,E1 25.1332,E2 -303.3988} C_DIS
LIN {X 39.374,Y 23.5257,Z 64,A 22.9388,B 24.8483,C -2.8413,E1 25.1389,E2 -299.5252} C_DIS
LIN {X 41.2674,Y 20.018,Z 64,A 18.1107,B 24.8495,C -2.8306,E1 25.1451,E2 -294.6975} C_DIS
LIN {X 42.3522,Y 17.6085,Z 64,A 15.2349,B 24.8496,C -2.8291,E1 25.1482,E2 -291.8338} C_DIS
LIN {X 43.065,Y 15.785,Z 64,A 12.8325,B 24.8503,C -2.8229,E1 25.1506,E2 -289.4301} C_DIS
LIN {X 43.6393,Y 14.1196,Z 64,A 10.753,B 24.8507,C -2.8187,E1 25.1525,E2 -287.3524} C_DIS
LIN {X 44.4922,Y 11.1453,Z 64,A 5.9316,B 24.8538,C -2.7897,E1 25.156,E2 -282.49} C_DIS
LIN {X 45.1439,Y 8.1102,Z 64,A 2.7608,B 24.8537,C -2.7909,E1 25.1576,E2 -279.3406} C_DIS
LIN {X 45.6093,Y 4.8505,Z 64,A -1.8445,B 24.856,C -2.7691,E1 25.1592,E2 -274.7109} C_DIS
LIN {X 45.8417,Y 1.5115,Z 64,A -5.3017,B 24.856,C -2.7695,E1 25.1597,E2 -271.2751} C_DIS
LIN {X 45.8648,Y -0.467,Z 64,A -8.4837,B 24.8581,C -2.7485,E1 25.1597,E2 -268.0624} C_DIS
LIN {X 45.7069,Y -3.8277,Z 64,A -12.7728,B 24.8596,C -2.7337,E1 25.1588,E2 -263.7638} C_DIS
LIN {X 45.3349,Y -6.964,Z 64,A -15.6802,B 24.8589,C -2.7406,E1 25.1577,E2 -260.8898} C_DIS
LIN {X 44.9583,Y -9.0839,Z 64,A -18.7975,B 24.8606,C -2.7242,E1 25.1561,E2 -257.752} C_DIS
LIN {X 44.488,Y -11.1621,Z 64,A -20.9937,B 24.8606,C -2.7246,E1 25.1547,E2 -255.5695} C_DIS
LIN {X 43.8702,Y -13.3845,Z 64,A -24.4299,B 24.8625,C -2.7054,E1 25.152,E2 -252.1075} C_DIS
LIN {X 42.9193,Y -16.1767,Z 64,A -28.2089,B 24.8639,C -2.6925,E1 25.1484,E2 -248.3192} C_DIS
LIN {X 41.4028,Y -19.7368,Z 64,A -32.3715,B 24.864,C -2.6906,E1 25.1437,E2 -244.1747} C_DIS
LIN {X 39.575,Y -23.1861,Z 64,A -36.9697,B 24.8649,C -2.6818,E1 25.1376,E2 -239.5798} C_DIS
LIN {X 38.6817,Y -24.6472,Z 64,A -39.5224,B 24.8663,C -2.6682,E1 25.1338,E2 -237.0079} C_DIS
LIN {X 37.4756,Y -26.4456,Z 64,A -42.1492,B 24.8669,C -2.6623,E1 25.1297,E2 -234.38} C_DIS
LIN {X 35.9802,Y -28.446,Z 64,A -45.5525,B 24.8682,C -2.6489,E1 25.1239,E2 -230.9612} C_DIS
LIN {X 34.4969,Y -30.2278,Z 64,A -48.0233,B 24.8682,C -2.6493,E1 25.1194,E2 -228.5025} C_DIS
LIN {X 33.3098,Y -31.5313,Z 64,A -50.2294,B 24.8688,C -2.6438,E1 25.1152,E2 -226.2931} C_DIS
LIN {X 31.5735,Y -33.2702,Z 64,A -53.7566,B 24.8703,C -2.6284,E1 25.1081,E2 -222.7441} C_DIS
LIN {X 29.7687,Y -34.8938,Z 64,A -56.2806,B 24.8701,C -2.6306,E1 25.1028,E2 -220.2354} C_DIS
LIN {X 28.4198,Y -36.0009,Z 64,A -58.4133,B 24.8704,C -2.6268,E1 25.0982,E2 -218.1017} C_DIS
LIN {X 26.5914,Y -37.3718,Z 64,A -61.6578,B 24.8717,C -2.6141,E1 25.0909,E2 -214.8387} C_DIS
LIN {X 24.5847,Y -38.7213,Z 64,A -64.5152,B 24.872,C -2.6112,E1 25.0842,E2 -211.9838} C_DIS
LIN {X 21.8554,Y -40.3248,Z 64,A -68.5319,B 24.8728,C -2.6032,E1 25.0744,E2 -207.9601} C_DIS
LIN {X 19.0481,Y -41.7244,Z 64,A -72.4987,B 24.8735,C -2.5962,E1 25.0644,E2 -203.9871} C_DIS
LIN {X 16.9466,Y -42.6211,Z 64,A -76.3558,B 24.8755,C -2.5755,E1 25.0543,E2 -200.0895} C_DIS
LIN {X 13.774,Y -43.7495,Z 64,A -80.0599,B 24.8752,C -2.5788,E1 25.0445,E2 -196.4002} C_DIS
LIN {X 9.7338,Y -44.8219,Z 64,A -84.4549,B 24.8743,C -2.5873,E1 25.0327,E2 -192.0319} C_DIS
LIN {X 7.8299,Y -45.193,Z 64,A -87.0031,B 24.8747,C -2.5833,E1 25.0257,E2 -189.4771} C_DIS
LIN {X 5.5797,Y -45.5262,Z 64,A -90.2535,B 24.8755,C -2.5749,E1 25.0166,E2 -186.2094} C_DIS
LIN {X 1.7385,Y -45.8341,Z 64,A -94.3572,B 24.8746,C -2.5842,E1 25.0052,E2 -182.1294} C_DIS
LIN {X 0.2949,Y -45.8474,Z 64,A -96.4193,B 24.875,C -2.5799,E1 24.9995,E2 -180.0574} C_DIS
Enddeposition()
LIN {X 0.2949,Y -45.8474,Z 64,A -96.4193,B 24.875,C -2.5799,E1 24.9995,E2 -180.0574} C_DIS
Startdeposition()
$VEL.CP = VEL_PRINT
LIN {X 0.3744,Y -44.9265,Z 64,A -94.9095,B 24.8713,C -2.6181,E1 25.0039,E2 -181.6579} C_DIS
LIN {X 2.7497,Y -44.8434,Z 64,A -91.839,B 24.8711,C -2.6199,E1 25.0125,E2 -184.7316} C_DIS
LIN {X 5.4133,Y -44.6009,Z 64,A -88.7779,B 24.8715,C -2.6161,E1 25.021,E2 -187.7817} C_DIS
LIN {X 6.9676,Y -44.3845,Z 64,A -86.4066,B 24.8708,C -2.6235,E1 25.0276,E2 -190.1685} C_DIS
LIN {X 9.5676,Y -43.8974,Z 64,A -82.9038,B 24.8703,C -2.6285,E1 25.0372,E2 -193.6788} C_DIS
LIN {X 12.9001,Y -43.0359,Z 64,A -79.0674,B 24.8707,C -2.6239,E1 25.0475,E2 -197.4981} C_DIS
LIN {X 14.6528,Y -42.4716,Z 64,A -76.5523,B 24.8702,C -2.6296,E1 25.0541,E2 -200.0217} C_DIS
LIN {X 17.3456,Y -41.4447,Z 64,A -72.8944,B 24.8697,C -2.6343,E1 25.0636,E2 -203.6826} C_DIS
LIN {X 19.1164,Y -40.6583,Z 64,A -70.2847,B 24.8691,C -2.6404,E1 25.0703,E2 -206.3003} C_DIS
LIN {X 21.675,Y -39.3543,Z 64,A -66.5433,B 24.8683,C -2.6479,E1 25.0795,E2 -210.0489} C_DIS
LIN {X 23.7303,Y -38.1496,Z 64,A -63.8032,B 24.8683,C -2.6482,E1 25.0861,E2 -212.7812} C_DIS
LIN {X 25.2483,Y -37.1623,Z 64,A -61.3739,B 24.8677,C -2.6548,E1 25.0917,E2 -215.218} C_DIS
LIN {X 27.0987,Y -35.8358,Z 64,A -58.5195,B 24.8672,C -2.6598,E1 25.0982,E2 -218.0742} C_DIS
LIN {X 29.0583,Y -34.2658,Z 64,A -54.4692,B 24.8649,C -2.682,E1 25.1069,E2 -222.1615} C_DIS
LIN {X 32.5387,Y -30.9804,Z 64,A -49.6354,B 24.8658,C -2.6735,E1 25.1165,E2 -226.9548} C_DIS
LIN {X 33.6806,Y -29.7347,Z 64,A -47.1536,B 24.8646,C -2.6847,E1 25.1212,E2 -229.4523} C_DIS
LIN {X 35.1278,Y -28.0106,Z 64,A -44.165,B 24.8637,C -2.6942,E1 25.1265,E2 -232.4496} C_DIS
LIN {X 36.6359,Y -26.0066,Z 64,A -40.9202,B 24.8627,C -2.7036,E1 25.1318,E2 -235.7009} C_DIS
LIN {X 37.8937,Y -24.1373,Z 64,A -38.2989,B 24.8624,C -2.7069,E1 25.1358,E2 -238.3168} C_DIS
LIN {X 38.879,Y -22.516,Z 64,A -35.8669,B 24.8617,C -2.714,E1 25.1393,E2 -240.753} C_DIS
LIN {X 40.2838,Y -19.8929,Z 64,A -32.5012,B 24.8614,C -2.717,E1 25.1436,E2 -244.1082} C_DIS
LIN {X 41.1865,Y -17.9498,Z 64,A -29.0446,B 24.8592,C -2.7385,E1 25.1476,E2 -247.5968} C_DIS
LIN {X 42.2331,Y -15.3261,Z 64,A -25.1428,B 24.8574,C -2.7549,E1 25.1515,E2 -251.5158} C_DIS
LIN {X 43.3955,Y -11.634,Z 64,A -20.9073,B 24.8572,C -2.757,E1 25.1548,E2 -255.7319} C_DIS
LIN {X 43.883,Y -9.6326,Z 64,A -18.2283,B 24.8563,C -2.7661,E1 25.1565,E2 -258.417} C_DIS
LIN {X 44.296,Y -7.5096,Z 64,A -15.0728,B 24.8546,C -2.7822,E1 25.158,E2 -261.5921} C_DIS
LIN {X 44.7781,Y -3.6669,Z 64,A -10.9271,B 24.8546,C -2.7829,E1 25.1593,E2 -265.7148} C_DIS
LIN {X 44.9025,Y -1.5045,Z 64,A -7.786,B 24.8529,C -2.7986,E1 25.1597,E2 -268.8746} C_DIS
LIN {X 44.9177,Y 0.9608,Z 64,A -4.5929,B 24.8517,C -2.8094,E1 25.1597,E2 -272.0741} C_DIS
LIN {X 44.7865,Y 3.5619,Z 64,A -1.3211,B 24.8507,C -2.8188,E1 25.1591,E2 -275.3488} C_DIS
LIN {X 44.5221,Y 6.0248,Z 64,A 1.5991,B 24.8502,C -2.8242,E1 25.1581,E2 -278.2644} C_DIS
LIN {X 44.2138,Y 7.9788,Z 64,A 4.1831,B 24.8492,C -2.833,E1 25.1569,E2 -280.8542} C_DIS
LIN {X 43.8022,Y 9.9953,Z 64,A 6.7186,B 24.8485,C -2.8393,E1 25.1554,E2 -283.3898} C_DIS
LIN {X 43.3495,Y 11.8044,Z 64,A 9.1569,B 24.8477,C -2.8475,E1 25.1537,E2 -285.8334} C_DIS
LIN {X 42.6465,Y 14.136,Z 64,A 12.4019,B 24.8464,C -2.8592,E1 25.1509,E2 -289.0877} C_DIS
LIN {X 41.7937,Y 16.4866,Z 64,A 15.175,B 24.8462,C -2.8607,E1 25.1482,E2 -291.8489} C_DIS
LIN {X 41.2684,Y 17.7614,Z 64,A 17.3305,B 24.8449,C -2.8729,E1 25.1458,E2 -294.0214} C_DIS
LIN {X 40.1333,Y 20.1951,Z 64,A 20.749,B 24.8439,C -2.8821,E1 25.1417,E2 -297.4435} C_DIS
LIN {X 39.0781,Y 22.169,Z 64,A 23.542,B 24.8432,C -2.8886,E1 25.1379,E2 -300.2372} C_DIS
LIN {X 37.7893,Y 24.3001,Z 64,A 26.7029,B 24.8424,C -2.8964,E1 25.1332,E2 -303.4006} C_DIS
LIN {X 36.4007,Y 26.3356,Z 64,A 29.7387,B 24.8417,C -2.9022,E1 25.1283,E2 -306.4353} C_DIS
LIN {X 34.8426,Y 28.3641,Z 64,A 32.8837,B 24.8411,C -2.9077,E1 25.1229,E2 -309.5787} C_DIS
LIN {X 33.4504,Y 29.9932,Z 64,A 35.9598,B 24.8398,C -2.9199,E1 25.1172,E2 -312.6698} C_DIS
LIN {X 30.9508,Y 32.5671,Z 64,A 40.7578,B 24.8383,C -2.9332,E1 25.1077,E2 -317.4792} C_DIS
LIN {X 28.3262,Y 34.8733,Z 64,A 44.634,B 24.8385,C -2.9315,E1 25.0994,E2 -321.3363} C_DIS
LIN {X 26.4888,Y 36.2887,Z 64,A 47.692,B 24.8378,C -2.9383,E1 25.0926,E2 -324.3994} C_DIS
LIN {X 24.444,Y 37.6968,Z 64,A 51.1012,B 24.8367,C -2.9474,E1 25.0846,E2 -327.8189} C_DIS
LIN {X 22.4139,Y 38.9376,Z 64,A 54.0467,B 24.8364,C -2.9502,E1 25.0776,E2 -330.7621} C_DIS
LIN {X 20.0834,Y 40.1896,Z 64,A 57.135,B 24.8364,C -2.9498,E1 25.0699,E2 -333.8406} C_DIS
LIN {X 18.0931,Y 41.1238,Z 64,A 60.0311,B 24.836,C -2.9544,E1 25.0626,E2 -336.7405} C_DIS
LIN {X 15.6113,Y 42.1286,Z 64,A 63.0913,B 24.8362,C -2.9519,E1 25.0546,E2 -339.7881} C_DIS
LIN {X 13.5141,Y 42.8471,Z 64,A 66.0514,B 24.8358,C -2.9563,E1 25.0468,E2 -342.753} C_DIS
LIN {X 11.8248,Y 43.344,Z 64,A 68.4748,B 24.8353,C -2.9607,E1 25.0402,E2 -345.1826} C_DIS
LIN {X 9.5051,Y 43.911,Z 64,A 71.1768,B 24.8357,C -2.9568,E1 25.0329,E2 -347.8717} C_DIS
LIN {X 8.2099,Y 44.1712,Z 64,A 72.9825,B 24.8354,C -2.9594,E1 25.028,E2 -349.6815} C_DIS
LIN {X 6.5869,Y 44.443,Z 64,A 75.2507,B 24.835,C -2.9626,E1 25.0217,E2 -351.9552} C_DIS
LIN {X 4.3208,Y 44.7196,Z 64,A 78.1244,B 24.835,C -2.9626,E1 25.0137,E2 -354.8266} C_DIS
LIN {X 1.9234,Y 44.8865,Z 64,A 81.2201,B 24.835,C -2.9629,E1 25.0051,E2 -357.9222} C_DIS
LIN {X -0.7693,Y 44.9213,Z 64,A 85.0385,B 24.8344,C -2.9681,E1 24.9944,E2 -361.7526} C_DIS
LIN {X -3.7572,Y 44.7707,Z 64,A 88.5481,B 24.8351,C -2.9619,E1 24.9847,E2 -365.2489} C_DIS
LIN {X -6.1015,Y 44.5121,Z 64,A 91.5783,B 24.8353,C -2.9605,E1 24.9763,E2 -368.2779} C_DIS
LIN {X -8.5954,Y 44.0981,Z 64,A 95.2964,B 24.8347,C -2.9653,E1 24.966,E2 -372.0113} C_DIS
LIN {X -12.2663,Y 43.2211,Z 64,A 99.5219,B 24.8362,C -2.9522,E1 24.9547,E2 -376.2117} C_DIS
LIN {X -14.363,Y 42.5701,Z 64,A 102.2871,B 24.8366,C -2.9485,E1 24.9473,E2 -378.973} C_DIS
LIN {X -16.2587,Y 41.8833,Z 64,A 104.9093,B 24.8369,C -2.9459,E1 24.9405,E2 -381.5944} C_DIS
LIN {X -18.274,Y 41.0433,Z 64,A 107.859,B 24.8371,C -2.9442,E1 24.9329,E2 -384.5472} C_DIS
LIN {X -20.1914,Y 40.1352,Z 64,A 110.9661,B 24.837,C -2.9455,E1 24.9251,E2 -387.6656} C_DIS
LIN {X -23.6349,Y 38.2092,Z 64,A 115.2156,B 24.8391,C -2.9261,E1 24.9149,E2 -391.8814} C_DIS
LIN {X -25.859,Y 36.7406,Z 64,A 119.6646,B 24.8383,C -2.9336,E1 24.9046,E2 -396.3633} C_DIS
LIN {X -28.7431,Y 34.5305,Z 64,A 124.0553,B 24.8397,C -2.9206,E1 24.8951,E2 -400.7393} C_DIS
LIN {X -31.354,Y 32.1787,Z 64,A 127.9035,B 24.8417,C -2.9021,E1 24.8873,E2 -404.5591} C_DIS
LIN {X -32.4868,Y 31.0346,Z 64,A 130.5158,B 24.8415,C -2.9044,E1 24.8822,E2 -407.1881} C_DIS
LIN {X -35.0674,Y 28.0867,Z 64,A 135.0413,B 24.8435,C -2.8858,E1 24.874,E2 -411.6897} C_DIS
LIN {X -36.7123,Y 25.8986,Z 64,A 139.0499,B 24.8438,C -2.8831,E1 24.8674,E2 -415.7113} C_DIS
LIN {X -38.2347,Y 23.594,Z 64,A 142.8853,B 24.8444,C -2.8773,E1 24.8617,E2 -419.5525} C_DIS
LIN {X -40.2719,Y 19.917,Z 64,A 147.6254,B 24.8469,C -2.8542,E1 24.8556,E2 -424.2624} C_DIS
LIN {X -41.5653,Y 17.0536,Z 64,A 151.6372,B 24.8482,C -2.8424,E1 24.8511,E2 -428.2682} C_DIS
LIN {X -42.382,Y 14.9094,Z 64,A 154.6318,B 24.8491,C -2.8345,E1 24.8482,E2 -431.2606} C_DIS
LIN {X -43.299,Y 11.9878,Z 64,A 159.081,B 24.8496,C -2.8292,E1 24.8447,E2 -435.7229} C_DIS
LIN {X -44.1742,Y 8.1978,Z 64,A 163.1522,B 24.8524,C -2.8029,E1 24.8423,E2 -439.7551} C_DIS
LIN {X -44.4832,Y 6.3058,Z 64,A 166.1153,B 24.8526,C -2.8015,E1 24.8411,E2 -442.7327} C_DIS
LIN {X -44.7293,Y 4.2205,Z 64,A 168.5076,B 24.8538,C -2.7897,E1 24.8404,E2 -445.1108} C_DIS
LIN {X -44.8611,Y 2.45,Z 64,A 170.8406,B 24.8545,C -2.7834,E1 24.8399,E2 -447.4429} C_DIS
LIN {X -44.9265,Y 0.4113,Z 64,A 173.6514,B 24.8551,C -2.7778,E1 24.8398,E2 -450.2572} C_DIS
LIN {X -44.9009,Y -1.5663,Z 64,A 175.9999,B 24.8561,C -2.7678,E1 24.8399,E2 -452.5959} C_DIS
LIN {X -44.8064,Y -3.312,Z 64,A 178.2935,B 24.8568,C -2.7616,E1 24.8404,E2 -454.8886} C_DIS
LIN {X -44.5411,Y -5.8827,Z 64,A -178.5886,B 24.858,C -2.7493,E1 24.8413,E2 -457.9955} C_DIS
LIN {X -44.0878,Y -8.6491,Z 64,A -174.5544,B 24.8586,C -2.744,E1 24.8433,E2 -462.041} C_DIS
LIN {X -43.5333,Y -11.1077,Z 64,A -170.9438,B 24.8591,C -2.7393,E1 24.8457,E2 -465.6616} C_DIS
LIN {X -42.3825,Y -14.9079,Z 64,A -166.8196,B 24.8618,C -2.7128,E1 24.8491,E2 -469.7459} C_DIS
LIN {X -41.5653,Y -17.0523,Z 64,A -163.1622,B 24.8618,C -2.7136,E1 24.8529,E2 -473.4259} C_DIS
LIN {X -40.2372,Y -19.9861,Z 64,A -158.704,B 24.8624,C -2.7068,E1 24.8583,E2 -477.8921} C_DIS
LIN {X -37.7004,Y -24.4385,Z 64,A -153.0277,B 24.8652,C -2.6788,E1 24.8663,E2 -483.5308} C_DIS
LIN {X -36.5114,Y -26.1811,Z 64,A -149.5402,B 24.8649,C -2.6826,E1 24.8719,E2 -487.0445} C_DIS
LIN {X -34.8446,Y -28.3616,Z 64,A -146.7615,B 24.8666,C -2.665,E1 24.8766,E2 -489.7942} C_DIS
LIN {X -32.9475,Y -30.5455,Z 64,A -142.1845,B 24.8663,C -2.6687,E1 24.8852,E2 -494.4005} C_DIS
LIN {X -30.6652,Y -32.8352,Z 64,A -138.9626,B 24.8683,C -2.6482,E1 24.8916,E2 -497.5869} C_DIS
LIN {X -29.7053,Y -33.7064,Z 64,A -136.9656,B 24.8682,C -2.6497,E1 24.8958,E2 -499.5954} C_DIS
LIN {X -27.7935,Y -35.2994,Z 64,A -133.4396,B 24.8682,C -2.6488,E1 24.9035,E2 -503.1325} C_DIS
LIN {X -25.1775,Y -37.2104,Z 64,A -129.6216,B 24.8694,C -2.6377,E1 24.9122,E2 -506.9372} C_DIS
LIN {X -22.7509,Y -38.7419,Z 64,A -125.9424,B 24.8699,C -2.6327,E1 24.9209,E2 -510.6158} C_DIS
LIN {X -20.6106,Y -39.9219,Z 64,A -122.6601,B 24.87,C -2.6311,E1 24.929,E2 -513.9035} C_DIS
LIN {X -18.4463,Y -40.9665,Z 64,A -120.1098,B 24.8711,C -2.6202,E1 24.9354,E2 -516.4343} C_DIS
LIN {X -16.59,Y -41.7524,Z 64,A -117.3175,B 24.8711,C -2.6209,E1 24.9426,E2 -519.2345} C_DIS
LIN {X -14.8755,Y -42.3938,Z 64,A -114.7868,B 24.8709,C -2.6218,E1 24.9493,E2 -521.7724} C_DIS
LIN {X -12.5436,Y -43.1412,Z 64,A -111.9779,B 24.8716,C -2.6149,E1 24.9568,E2 -524.5699} C_DIS
LIN {X -11.14,Y -43.5248,Z 64,A -110.0507,B 24.8716,C -2.6149,E1 24.962,E2 -526.4999} C_DIS
LIN {X -9.6585,Y -43.8776,Z 64,A -107.7751,B 24.8712,C -2.619,E1 24.9682,E2 -528.7881} C_DIS
LIN {X -6.5718,Y -44.4452,Z 64,A -103.6536,B 24.8712,C -2.6196,E1 24.9796,E2 -532.9151} C_DIS
LIN {X -3.9829,Y -44.751,Z 64,A -99.9911,B 24.8707,C -2.6247,E1 24.9898,E2 -536.5915} C_DIS
LIN {X 0.3111,Y -44.9254,Z 64,A -97.1276,B 24.8746,C -2.5847,E1 24.9975,E2 -539.3607} C_DIS
Enddeposition()
LIN {X 0.3111,Y -44.9254,Z 64,A -97.1276,B 24.8746,C -2.5847,E1 24.9975,E2 -539.3607} C_DIS
Startdeposition()
$VEL.CP = VEL_PRINT
LIN {X -0.4192,Y -43.9874,Z 64,A -97.8588,B 24.8726,C -2.6044,E1 24.9956,E2 -538.6762} C_DIS
LIN {X -3.79,Y -43.8256,Z 64,A -101.8099,B 24.872,C -2.6109,E1 24.9846,E2 -534.7392} C_DIS
LIN {X -6.0232,Y -43.5752,Z 64,A -104.6303,B 24.8718,C -2.6129,E1 24.9768,E2 -531.9217} C_DIS
LIN {X -7.7859,Y -43.2947,Z 64,A -106.9787,B 24.8718,C -2.6133,E1 24.9704,E2 -529.5718} C_DIS
LIN {X -9.5057,Y -42.9501,Z 64,A -109.2849,B 24.8718,C -2.614,E1 24.9641,E2 -527.2645} C_DIS
LIN {X -11.3424,Y -42.5014,Z 64,A -111.8233,B 24.8717,C -2.6142,E1 24.9572,E2 -524.723} C_DIS
LIN {X -13.3225,Y -41.923,Z 64,A -114.3644,B 24.8713,C -2.6182,E1 24.9504,E2 -522.187} C_DIS
LIN {X -15.7829,Y -41.0602,Z 64,A -118.5398,B 24.8721,C -2.6103,E1 24.9394,E2 -517.9844} C_DIS
LIN {X -19.5847,Y -39.3884,Z 64,A -123.7228,B 24.8712,C -2.6195,E1 24.9263,E2 -512.8102} C_DIS
LIN {X -21.7333,Y -38.2459,Z 64,A -126.3912,B 24.8701,C -2.6303,E1 24.9198,E2 -510.1601} C_DIS
LIN {X -24.1955,Y -36.7373,Z 64,A -129.815,B 24.8691,C -2.6404,E1 24.9117,E2 -506.7495} C_DIS
LIN {X -25.8124,Y -35.6205,Z 64,A -133.1898,B 24.8697,C -2.6338,E1 24.904,E2 -503.3474} C_DIS
LIN {X -27.9036,Y -34.0072,Z 64,A -136.2126,B 24.8686,C -2.6453,E1 24.8974,E2 -500.3409} C_DIS
LIN {X -29.081,Y -33.0057,Z 64,A -138.4209,B 24.8685,C -2.6466,E1 24.8927,E2 -498.1269} C_DIS
LIN {X -31.1182,Y -31.0929,Z 64,A -142.3946,B 24.8682,C -2.6497,E1 24.8847,E2 -494.1442} C_DIS
LIN {X -33.4816,Y -28.5313,Z 64,A -147.0077,B 24.8673,C -2.6588,E1 24.8762,E2 -489.5321} C_DIS
LIN {X -35.674,Y -25.7383,Z 64,A -151.6926,B 24.8662,C -2.6691,E1 24.8683,E2 -484.8493} C_DIS
LIN {X -36.8587,Y -24.0109,Z 64,A -154.7257,B 24.8659,C -2.6722,E1 24.8637,E2 -481.8085} C_DIS
LIN {X -38.5837,Y -21.1277,Z 64,A -158.4261,B 24.8639,C -2.6918,E1 24.8586,E2 -478.1354} C_DIS
LIN {X -39.6087,Y -19.1366,Z 64,A -161.0896,B 24.8628,C -2.7027,E1 24.8553,E2 -475.4838} C_DIS
LIN {X -40.2377,Y -17.7758,Z 64,A -163.4323,B 24.8628,C -2.7035,E1 24.8526,E2 -473.1301} C_DIS
LIN {X -41.4138,Y -14.8301,Z 64,A -167.1786,B 24.8611,C -2.7198,E1 24.8488,E2 -469.4017} C_DIS
LIN {X -41.9185,Y -13.3373,Z 64,A -169.3401,B 24.8606,C -2.7245,E1 24.8469,E2 -467.2391} C_DIS
LIN {X -42.4429,Y -11.56,Z 64,A -172.1878,B 24.8604,C -2.7265,E1 24.8448,E2 -464.3799} C_DIS
LIN {X -43.0853,Y -8.8718,Z 64,A -175.9654,B 24.8595,C -2.7353,E1 24.8425,E2 -460.6011} C_DIS
LIN {X -43.5626,Y -6.1123,Z 64,A -179.1232,B 24.8577,C -2.7522,E1 24.8411,E2 -457.4647} C_DIS
LIN {X -43.7668,Y -4.4183,Z 64,A 178.323,B 24.8574,C -2.7552,E1 24.8404,E2 -454.9029} C_DIS
LIN {X -43.9624,Y -1.5317,Z 64,A 174.8288,B 24.8559,C -2.7701,E1 24.8398,E2 -451.4234} C_DIS
LIN {X -43.9825,Y 0.7444,Z 64,A 171.6702,B 24.8551,C -2.7772,E1 24.8398,E2 -448.2626} C_DIS
LIN {X -43.8799,Y 3.1015,Z 64,A 168.6691,B 24.854,C -2.7877,E1 24.8403,E2 -445.2685} C_DIS
LIN {X -43.6796,Y 5.211,Z 64,A 165.9885,B 24.853,C -2.7972,E1 24.8411,E2 -442.5948} C_DIS
LIN {X -43.425,Y 7.0268,Z 64,A 163.3844,B 24.8525,C -2.8022,E1 24.8422,E2 -439.9871} C_DIS
LIN {X -42.9802,Y 9.3676,Z 64,A 159.4245,B 24.8525,C -2.8022,E1 24.8445,E2 -436.0037} C_DIS
LIN {X -42.0327,Y 12.9719,Z 64,A 155.4406,B 24.8499,C -2.827,E1 24.8475,E2 -432.0561} C_DIS
LIN {X -41.304,Y 15.1333,Z 64,A 152.7148,B 24.8486,C -2.8388,E1 24.85,E2 -429.3431} C_DIS
LIN {X -40.5536,Y 17.043,Z 64,A 149.6719,B 24.8482,C -2.8425,E1 24.8532,E2 -426.292} C_DIS
LIN {X -39.6889,Y 18.9694,Z 64,A 147.1573,B 24.847,C -2.8533,E1 24.8561,E2 -423.7896} C_DIS
LIN {X -38.5077,Y 21.2657,Z 64,A 143.0949,B 24.8469,C -2.8547,E1 24.8615,E2 -419.709} C_DIS
LIN {X -37.166,Y 23.5324,Z 64,A 139.5266,B 24.846,C -2.8626,E1 24.8668,E2 -416.1414} C_DIS
LIN {X -34.753,Y 26.9687,Z 64,A 134.3715,B 24.8441,C -2.8808,E1 24.8752,E2 -411.0048} C_DIS
LIN {X -33.2221,Y 28.8327,Z 64,A 131.393,B 24.843,C -2.8906,E1 24.8806,E2 -408.0362} C_DIS
LIN {X -31.2943,Y 30.9147,Z 64,A 127.0212,B 24.843,C -2.8913,E1 24.8891,E2 -403.6473} C_DIS
LIN {X -28.087,Y 33.8549,Z 64,A 122.3827,B 24.8402,C -2.9166,E1 24.8987,E2 -399.0508} C_DIS
LIN {X -25.7164,Y 35.6898,Z 64,A 117.3922,B 24.8408,C -2.911,E1 24.9099,E2 -394.0289} C_DIS
LIN {X -23.3932,Y 37.2535,Z 64,A 113.9044,B 24.8398,C -2.9197,E1 24.9181,E2 -390.5509} C_DIS
LIN {X -20.028,Y 39.1653,Z 64,A 109.668,B 24.8377,C -2.9386,E1 24.9284,E2 -386.3473} C_DIS
LIN {X -18.764,Y 39.7863,Z 64,A 107.5327,B 24.8379,C -2.9374,E1 24.9338,E2 -384.2038} C_DIS
LIN {X -16.5166,Y 40.7707,Z 64,A 104.771,B 24.8367,C -2.9477,E1 24.9408,E2 -381.4602} C_DIS
LIN {X -14.7814,Y 41.4313,Z 64,A 101.8369,B 24.8371,C -2.9438,E1 24.9485,E2 -378.5109} C_DIS
LIN {X -12.8339,Y 42.0753,Z 64,A 99.4864,B 24.8363,C -2.9512,E1 24.9548,E2 -376.1738} C_DIS
LIN {X -10.3967,Y 42.7428,Z 64,A 95.4216,B 24.8371,C -2.9439,E1 24.9658,E2 -372.0856} C_DIS
LIN {X -7.8011,Y 43.292,Z 64,A 92.2976,B 24.8363,C -2.9511,E1 24.9743,E2 -368.9754} C_DIS
LIN {X -5.1642,Y 43.6851,Z 64,A 89.1905,B 24.8355,C -2.9584,E1 24.9829,E2 -365.8833} C_DIS
LIN {X -3.5043,Y 43.8494,Z 64,A 86.9733,B 24.8355,C -2.9588,E1 24.9891,E2 -363.6658} C_DIS
LIN {X -1.7095,Y 43.9563,Z 64,A 84.4576,B 24.8357,C -2.9571,E1 24.9961,E2 -361.1455} C_DIS
LIN {X 0.6148,Y 43.985,Z 64,A 81.6274,B 24.8353,C -2.9605,E1 25.004,E2 -358.3236} C_DIS
LIN {X 2.3615,Y 43.9259,Z 64,A 79.3906,B 24.8353,C -2.9612,E1 25.0102,E2 -356.0891} C_DIS
LIN {X 4.0134,Y 43.8058,Z 64,A 76.7871,B 24.836,C -2.9545,E1 25.0175,E2 -353.4712} C_DIS
LIN {X 6.4343,Y 43.5166,Z 64,A 73.2829,B 24.8366,C -2.9489,E1 25.0272,E2 -349.9566} C_DIS
LIN {X 9.35,Y 42.9841,Z 64,A 70.0871,B 24.8356,C -2.9572,E1 25.0359,E2 -346.7845} C_DIS
LIN {X 11.047,Y 42.5796,Z 64,A 67.3197,B 24.8366,C -2.9484,E1 25.0434,E2 -344.0003} C_DIS
LIN {X 14.5953,Y 41.4974,Z 64,A 63.3864,B 24.8355,C -2.9586,E1 25.0538,E2 -340.0984} C_DIS
LIN {X 16.9177,Y 40.6054,Z 64,A 59.3604,B 24.8372,C -2.9431,E1 25.0643,E2 -336.0447} C_DIS
LIN {X 19.7359,Y 39.3126,Z 64,A 55.2462,B 24.8379,C -2.9372,E1 25.0747,E2 -331.9271} C_DIS
LIN {X 21.9146,Y 38.1419,Z 64,A 51.6149,B 24.8391,C -2.9262,E1 25.0836,E2 -328.2806} C_DIS
LIN {X 24.7929,Y 36.3372,Z 64,A 47.7979,B 24.8388,C -2.9291,E1 25.0924,E2 -324.4831} C_DIS
LIN {X 27.1647,Y 34.5999,Z 64,A 44.4932,B 24.8386,C -2.9311,E1 25.0998,E2 -321.1951} C_DIS
LIN {X 29.183,Y 32.9148,Z 64,A 40.6992,B 24.8399,C -2.9185,E1 25.1078,E2 -317.3861} C_DIS
LIN {X 31.3068,Y 30.9021,Z 64,A 37.0148,B 24.8406,C -2.9129,E1 25.1152,E2 -313.7036} C_DIS
LIN {X 32.781,Y 29.3336,Z 64,A 33.7437,B 24.8421,C -2.8989,E1 25.1214,E2 -310.4138} C_DIS
LIN {X 35.0483,Y 26.584,Z 64,A 29.7,B 24.8421,C -2.8983,E1 25.1284,E2 -306.3875} C_DIS
LIN {X 36.1375,Y 25.0826,Z 64,A 27.3665,B 24.8427,C -2.8938,E1 25.1322,E2 -304.0548} C_DIS
LIN {X 37.106,Y 23.6268,Z 64,A 25.193,B 24.8431,C -2.8899,E1 25.1355,E2 -301.8829} C_DIS
LIN {X 37.8277,Y 22.4526,Z 64,A 22.7609,B 24.8448,C -2.8742,E1 25.139,E2 -299.4261} C_DIS
LIN {X 38.9382,Y 20.4661,Z 64,A 19.5399,B 24.8461,C -2.8618,E1 25.1433,E2 -296.1928} C_DIS
LIN {X 40.2067,Y 17.8454,Z 64,A 16.5901,B 24.8457,C -2.8661,E1 25.1467,E2 -293.269} C_DIS
LIN {X 40.8574,Y 16.3007,Z 64,A 13.6011,B 24.8479,C -2.8457,E1 25.1498,E2 -290.2484} C_DIS
LIN {X 41.8983,Y 13.4008,Z 64,A 10.083,B 24.8482,C -2.8428,E1 25.153,E2 -286.7431} C_DIS
LIN {X 42.6499,Y 10.7733,Z 64,A 6.9271,B 24.8485,C -2.8393,E1 25.1553,E2 -283.5972} C_DIS
LIN {X 43.0115,Y 9.2219,Z 64,A 4.9505,B 24.849,C -2.8348,E1 25.1565,E2 -281.6215} C_DIS
LIN {X 43.2837,Y 7.8474,Z 64,A 2.75,B 24.8503,C -2.8226,E1 25.1576,E2 -279.4047} C_DIS
LIN {X 43.681,Y 5.1994,Z 64,A -0.3949,B 24.8508,C -2.818,E1 25.1588,E2 -276.2675} C_DIS
LIN {X 43.8713,Y 3.222,Z 64,A -3.1888,B 24.8521,C -2.8062,E1 25.1595,E2 -273.4624} C_DIS
LIN {X 43.9761,Y 1.0763,Z 64,A -5.8553,B 24.8527,C -2.7998,E1 25.1598,E2 -270.7966} C_DIS
LIN {X 43.9761,Y -1.0721,Z 64,A -8.8276,B 24.854,C -2.7879,E1 25.1597,E2 -267.8138} C_DIS
LIN {X 43.8416,Y -3.6029,Z 64,A -12.0227,B 24.8549,C -2.7794,E1 25.1591,E2 -264.6176} C_DIS
LIN {X 43.5737,Y -6.0342,Z 64,A -15.3038,B 24.8561,C -2.7677,E1 25.1579,E2 -261.3282} C_DIS
LIN {X 43.2472,Y -8.0476,Z 64,A -17.6207,B 24.8563,C -2.7655,E1 25.1568,E2 -259.0196} C_DIS
LIN {X 42.7953,Y -10.1787,Z 64,A -20.7476,B 24.8578,C -2.7515,E1 25.1549,E2 -255.8778} C_DIS
LIN {X 42.0516,Y -12.9112,Z 64,A -24.6674,B 24.8594,C -2.736,E1 25.1519,E2 -251.9437} C_DIS
LIN {X 41.191,Y -15.4395,Z 64,A -28.0087,B 24.8602,C -2.7279,E1 25.1487,E2 -248.602} C_DIS
LIN {X 40.0284,Y -18.2418,Z 64,A -31.744,B 24.861,C -2.72,E1 25.1445,E2 -244.8685} C_DIS
LIN {X 39.1254,Y -20.1064,Z 64,A -34.7728,B 24.8624,C -2.7063,E1 25.1407,E2 -241.8234} C_DIS
LIN {X 37.4033,Y -23.1534,Z 64,A -38.974,B 24.8631,C -2.6998,E1 25.1348,E2 -237.6284} C_DIS
LIN {X 35.7904,Y -25.5754,Z 64,A -42.9668,B 24.8645,C -2.686,E1 25.1284,E2 -233.6224} C_DIS
LIN {X 34.289,Y -27.5562,Z 64,A -45.748,B 24.8645,C -2.6855,E1 25.1237,E2 -230.8531} C_DIS
LIN {X 33.0677,Y -29.0102,Z 64,A -48.3081,B 24.8654,C -2.6777,E1 25.119,E2 -228.2863} C_DIS
LIN {X 31.7506,Y -30.4461,Z 64,A -51.17,B 24.8665,C -2.6659,E1 25.1135,E2 -225.409} C_DIS
LIN {X 29.3852,Y -32.7348,Z 64,A -54.772,B 24.8664,C -2.6678,E1 25.1062,E2 -221.8262} C_DIS
LIN {X 27.9875,Y -33.9377,Z 64,A -57.4567,B 24.8674,C -2.6576,E1 25.1005,E2 -219.1279} C_DIS
LIN {X 26.4291,Y -35.1647,Z 64,A -59.8574,B 24.8676,C -2.6553,E1 25.0952,E2 -216.7305} C_DIS
LIN {X 25.0756,Y -36.1422,Z 64,A -61.9351,B 24.8679,C -2.6526,E1 25.0904,E2 -214.6536} C_DIS
LIN {X 23.957,Y -36.8937,Z 64,A -64.4819,B 24.8695,C -2.636,E1 25.0844,E2 -212.0757} C_DIS
LIN {X 21.2789,Y -38.5005,Z 64,A -68.649,B 24.8704,C -2.6272,E1 25.0743,E2 -207.9004} C_DIS
LIN {X 17.4483,Y -40.3811,Z 64,A -74.3682,B 24.8715,C -2.6162,E1 25.0597,E2 -202.1694} C_DIS
LIN {X 13.439,Y -41.8862,Z 64,A -78.8964,B 24.8705,C -2.626,E1 25.0479,E2 -197.6738} C_DIS
LIN {X 12.1154,Y -42.2875,Z 64,A -81.1574,B 24.8714,C -2.6167,E1 25.0418,E2 -195.3945} C_DIS
LIN {X 9.4014,Y -42.9728,Z 64,A -84.8798,B 24.8719,C -2.6121,E1 25.0317,E2 -191.6663} C_DIS
LIN {X 6.0936,Y -43.5652,Z 64,A -88.7865,B 24.8715,C -2.6162,E1 25.021,E2 -187.7734} C_DIS
LIN {X 3.7887,Y -43.8254,Z 64,A -91.8426,B 24.8717,C -2.614,E1 25.0125,E2 -184.7141} C_DIS
LIN {X 1.8901,Y -43.9486,Z 64,A -94.4262,B 24.872,C -2.6114,E1 25.0052,E2 -182.1252} C_DIS
LIN {X 0.3067,Y -43.9841,Z 64,A -95.94,B 24.8712,C -2.6192,E1 25.0011,E2 -180.6303} C_DIS
Enddeposition()
LIN {X 0.3067,Y -43.9841,Z 64,A -95.94,B 24.8712,C -2.6192,E1 25.0011,E2 -180.6303} C_DIS
Startdeposition()
$VEL.CP = VEL_PRINT
LIN {X 1.3466,Y -43.0295,Z 64,A -93.9733,B 24.8687,C -2.6446,E1 25.0067,E2 -182.6569} C_DIS
LIN {X 3.3924,Y -42.9167,Z 64,A -90.6457,B 24.8676,C -2.655,E1 25.0161,E2 -186.0078} C_DIS
LIN {X 7.3742,Y -42.414,Z 64,A -85.1879,B 24.8671,C -2.6605,E1 25.0311,E2 -191.4736} C_DIS
LIN {X 10.2385,Y -41.8153,Z 64,A -81.7838,B 24.8675,C -2.6563,E1 25.0404,E2 -194.863} C_DIS
LIN {X 12.3123,Y -41.2524,Z 64,A -79.0101,B 24.8673,C -2.658,E1 25.0478,E2 -197.6361} C_DIS
LIN {X 14.4263,Y -40.5613,Z 64,A -75.8731,B 24.8667,C -2.6645,E1 25.0561,E2 -200.7824} C_DIS
LIN {X 16.6432,Y -39.7034,Z 64,A -73.0344,B 24.8667,C -2.6636,E1 25.0635,E2 -203.6125} C_DIS
LIN {X 18.5227,Y -38.8616,Z 64,A -70.198,B 24.8662,C -2.6693,E1 25.0707,E2 -206.4553} C_DIS
LIN {X 20.1755,Y -38.0304,Z 64,A -67.6848,B 24.8657,C -2.6742,E1 25.0769,E2 -208.9732} C_DIS
LIN {X 21.938,Y -37.0414,Z 64,A -64.7711,B 24.8648,C -2.6827,E1 25.084,E2 -211.8982} C_DIS
LIN {X 24.1882,Y -35.6125,Z 64,A -61.621,B 24.8648,C -2.6827,E1 25.0913,E2 -215.0381} C_DIS
LIN {X 25.7596,Y -34.4936,Z 64,A -58.7784,B 24.8638,C -2.6927,E1 25.0978,E2 -217.8941} C_DIS
LIN {X 27.6334,Y -33.0115,Z 64,A -55.4409,B 24.8629,C -2.7023,E1 25.105,E2 -221.2415} C_DIS
LIN {X 29.1032,Y -31.723,Z 64,A -52.9291,B 24.8624,C -2.7066,E1 25.1102,E2 -223.7536} C_DIS
LIN {X 30.6351,Y -30.2463,Z 64,A -50.2954,B 24.8621,C -2.7099,E1 25.1154,E2 -226.384} C_DIS
LIN {X 32.1659,Y -28.6132,Z 64,A -47.6677,B 24.862,C -2.7112,E1 25.1203,E2 -229.0031} C_DIS
LIN {X 33.0495,Y -27.5878,Z 64,A -45.512,B 24.8609,C -2.7219,E1 25.1242,E2 -231.1744} C_DIS
LIN {X 34.9481,Y -25.1397,Z 64,A -40.897,B 24.8588,C -2.7415,E1 25.132,E2 -235.8137} C_DIS
LIN {X 36.4149,Y -22.9635,Z 64,A -37.6619,B 24.8583,C -2.7466,E1 25.1369,E2 -239.0445} C_DIS
LIN {X 38.0072,Y -20.2186,Z 64,A -33.6232,B 24.8574,C -2.7553,E1 25.1423,E2 -243.0829} C_DIS
LIN {X 38.8925,Y -18.458,Z 64,A -30.7463,B 24.8561,C -2.7675,E1 25.1458,E2 -245.9732} C_DIS
LIN {X 40.2592,Y -15.2495,Z 64,A -26.7774,B 24.8559,C -2.7693,E1 25.15,E2 -249.9245} C_DIS
LIN {X 40.794,Y -13.7546,Z 64,A -24.312,B 24.8546,C -2.7821,E1 25.1522,E2 -252.4062} C_DIS
LIN {X 41.5524,Y -11.2582,Z 64,A -20.7052,B 24.8532,C -2.7952,E1 25.155,E2 -256.0234} C_DIS
LIN {X 42.3198,Y -7.8967,Z 64,A -16.7085,B 24.8529,C -2.7988,E1 25.1573,E2 -260.0053} C_DIS
LIN {X 42.6666,Y -5.7356,Z 64,A -13.6871,B 24.8517,C -2.8099,E1 25.1586,E2 -263.0351} C_DIS
LIN {X 42.8836,Y -3.7871,Z 64,A -11.0311,B 24.8507,C -2.8189,E1 25.1593,E2 -265.6968} C_DIS
LIN {X 43.0228,Y -1.5426,Z 64,A -8.1321,B 24.8499,C -2.8267,E1 25.1597,E2 -268.5968} C_DIS
LIN {X 43.0497,Y 0.3308,Z 64,A -5.6994,B 24.8492,C -2.8334,E1 25.1597,E2 -271.031} C_DIS
LIN {X 43.0066,Y 1.9447,Z 64,A -3.4014,B 24.8482,C -2.8428,E1 25.1595,E2 -273.3376} C_DIS
LIN {X 42.8286,Y 4.363,Z 64,A -0.1498,B 24.847,C -2.8533,E1 25.1587,E2 -276.5947} C_DIS
LIN {X 42.5213,Y 6.7304,Z 64,A 2.8763,B 24.8463,C -2.8603,E1 25.1575,E2 -279.6197} C_DIS
LIN {X 42.1925,Y 8.5524,Z 64,A 5.2689,B 24.8456,C -2.8666,E1 25.1563,E2 -282.0131} C_DIS
LIN {X 41.7155,Y 10.6384,Z 64,A 8.2285,B 24.8445,C -2.8771,E1 25.1543,E2 -284.9804} C_DIS
LIN {X 41.1464,Y 12.6618,Z 64,A 11.188,B 24.8433,C -2.8882,E1 25.1519,E2 -287.9494} C_DIS
LIN {X 40.1708,Y 15.4804,Z 64,A 14.8165,B 24.8427,C -2.8936,E1 25.1485,E2 -291.5704} C_DIS
LIN {X 39.628,Y 16.8217,Z 64,A 17.1692,B 24.8413,C -2.9066,E1 25.1459,E2 -293.9407} C_DIS
LIN {X 38.2361,Y 19.7834,Z 64,A 21.0396,B 24.8409,C -2.9099,E1 25.1412,E2 -297.7984} C_DIS
LIN {X 37.2454,Y 21.5905,Z 64,A 24.2214,B 24.8393,C -2.9248,E1 25.1368,E2 -300.9988} C_DIS
LIN {X 35.7888,Y 23.9276,Z 64,A 27.5006,B 24.839,C -2.9273,E1 25.1319,E2 -304.2676} C_DIS
LIN {X 34.8072,Y 25.3342,Z 64,A 29.5951,B 24.8387,C -2.9297,E1 25.1285,E2 -306.3575} C_DIS
LIN {X 33.4471,Y 27.1042,Z 64,A 32.7779,B 24.8375,C -2.9402,E1 25.123,E2 -309.5504} C_DIS
LIN {X 32.1116,Y 28.674,Z 64,A 35.414,B 24.8371,C -2.9445,E1 25.1181,E2 -312.1849} C_DIS
LIN {X 30.6066,Y 30.2751,Z 64,A 38.7438,B 24.8356,C -2.9576,E1 25.1116,E2 -315.5312} C_DIS
LIN {X 27.4744,Y 33.1435,Z 64,A 43.8432,B 24.8354,C -2.9593,E1 25.101,E2 -320.6142} C_DIS
LIN {X 25.4544,Y 34.7192,Z 64,A 47.7944,B 24.8338,C -2.9741,E1 25.0922,E2 -324.5863} C_DIS
LIN {X 23.5169,Y 36.0602,Z 64,A 51.34,B 24.8325,C -2.9857,E1 25.0839,E2 -328.1477} C_DIS
LIN {X 21.0236,Y 37.5681,Z 64,A 54.5726,B 24.833,C -2.9806,E1 25.0761,E2 -331.3586} C_DIS
LIN {X 18.772,Y 38.7424,Z 64,A 57.8688,B 24.8327,C -2.9834,E1 25.0679,E2 -334.6525} C_DIS
LIN {X 16.798,Y 39.6381,Z 64,A 60.6823,B 24.8325,C -2.9854,E1 25.0607,E2 -337.464} C_DIS
LIN {X 14.5963,Y 40.5005,Z 64,A 63.4112,B 24.8329,C -2.9819,E1 25.0536,E2 -340.1784} C_DIS
LIN {X 12.9701,Y 41.0499,Z 64,A 66.2848,B 24.8317,C -2.9927,E1 25.0459,E2 -343.0725} C_DIS
LIN {X 10.2631,Y 41.8093,Z 64,A 69.8403,B 24.8317,C -2.9922,E1 25.0363,E2 -346.621} C_DIS
LIN {X 8.6033,Y 42.1822,Z 64,A 72.6239,B 24.8307,C -3.0011,E1 25.0287,E2 -349.4224} C_DIS
LIN {X 6.0625,Y 42.6215,Z 64,A 75.4777,B 24.8316,C -2.9934,E1 25.0209,E2 -352.2551} C_DIS
LIN {X 4.2034,Y 42.8447,Z 64,A 78.1779,B 24.8312,C -2.9968,E1 25.0134,E2 -354.9617} C_DIS
LIN {X 1.4447,Y 43.0262,Z 64,A 81.6431,B 24.8316,C -2.9935,E1 25.0037,E2 -358.418} C_DIS
LIN {X -0.2882,Y 43.0496,Z 64,A 83.7711,B 24.8319,C -2.9905,E1 24.9978,E2 -360.5387} C_DIS
LIN {X -2.1316,Y 42.9978,Z 64,A 86.4691,B 24.8316,C -2.9933,E1 24.9902,E2 -363.2437} C_DIS
LIN {X -4.2953,Y 42.8357,Z 64,A 89.3389,B 24.8318,C -2.9917,E1 24.9823,E2 -366.111} C_DIS
LIN {X -6.2086,Y 42.6006,Z 64,A 91.8138,B 24.8321,C -2.9888,E1 24.9754,E2 -368.5811} C_DIS
LIN {X -8.3451,Y 42.2342,Z 64,A 94.598,B 24.8325,C -2.9853,E1 24.9678,E2 -371.3596} C_DIS
LIN {X -9.7401,Y 41.9338,Z 64,A 96.7059,B 24.8324,C -2.9865,E1 24.962,E2 -373.4731} C_DIS
LIN {X -11.9323,Y 41.3637,Z 64,A 99.6436,B 24.8328,C -2.9824,E1 24.9541,E2 -376.4056} C_DIS
LIN {X -13.759,Y 40.7926,Z 64,A 102.2171,B 24.8331,C -2.9798,E1 24.9473,E2 -378.9776} C_DIS
LIN {X -15.2976,Y 40.241,Z 64,A 104.2238,B 24.8337,C -2.9748,E1 24.9421,E2 -380.9765} C_DIS
LIN {X -17.0173,Y 39.5447,Z 64,A 106.9901,B 24.8337,C -2.9753,E1 24.9349,E2 -383.7503} C_DIS
LIN {X -18.9778,Y 38.6417,Z 64,A 109.777,B 24.8342,C -2.9698,E1 24.9279,E2 -386.5311} C_DIS
LIN {X -21.2591,Y 37.4357,Z 64,A 113.676,B 24.8342,C -2.97,E1 24.9184,E2 -390.4419} C_DIS
LIN {X -23.6799,Y 35.9528,Z 64,A 117.416,B 24.8351,C -2.9626,E1 24.9096,E2 -394.1761} C_DIS
LIN {X -26.2668,Y 34.1087,Z 64,A 121.0762,B 24.8368,C -2.9469,E1 24.9014,E2 -397.8118} C_DIS
LIN {X -27.4201,Y 33.1888,Z 64,A 123.8052,B 24.8362,C -2.9522,E1 24.8955,E2 -400.5639} C_DIS
LIN {X -30.2424,Y 30.6389,Z 64,A 128.429,B 24.8381,C -2.9352,E1 24.8861,E2 -405.166} C_DIS
LIN {X -32.3225,Y 28.4363,Z 64,A 132.9185,B 24.8386,C -2.931,E1 24.8776,E2 -409.6651} C_DIS
LIN {X -34.0238,Y 26.377,Z 64,A 135.8973,B 24.8403,C -2.9149,E1 24.8725,E2 -412.6194} C_DIS
LIN {X -35.3743,Y 24.536,Z 64,A 139.3055,B 24.8408,C -2.9112,E1 24.8669,E2 -416.0354} C_DIS
LIN {X -36.5408,Y 22.7623,Z 64,A 141.6349,B 24.8422,C -2.8975,E1 24.8635,E2 -418.344} C_DIS
LIN {X -37.6711,Y 20.8389,Z 64,A 145.1728,B 24.8424,C -2.8959,E1 24.8585,E2 -421.8964} C_DIS
LIN {X -38.862,Y 18.5223,Z 64,A 148.4907,B 24.8437,C -2.8841,E1 24.8544,E2 -425.2039} C_DIS
LIN {X -39.756,Y 16.5178,Z 64,A 151.2756,B 24.8448,C -2.8739,E1 24.8514,E2 -427.9797} C_DIS
LIN {X -40.5705,Y 14.4006,Z 64,A 154.6127,B 24.8454,C -2.8685,E1 24.8482,E2 -431.3228} C_DIS
LIN {X -41.3137,Y 12.1042,Z 64,A 157.2216,B 24.8472,C -2.8517,E1 24.846,E2 -433.9066} C_DIS
LIN {X -41.7256,Y 10.5968,Z 64,A 159.7652,B 24.8473,C -2.8506,E1 24.8442,E2 -436.4624} C_DIS
LIN {X -42.2324,Y 8.3552,Z 64,A 162.7382,B 24.8485,C -2.8401,E1 24.8425,E2 -439.4279} C_DIS
LIN {X -42.5889,Y 6.29,Z 64,A 165.5077,B 24.8494,C -2.8312,E1 24.8413,E2 -442.1924} C_DIS
LIN {X -42.8616,Y 4.0263,Z 64,A 168.7331,B 24.8502,C -2.8239,E1 24.8403,E2 -445.4197} C_DIS
LIN {X -43.0247,Y 1.4852,Z 64,A 172.3399,B 24.8511,C -2.8158,E1 24.8398,E2 -449.0287} C_DIS
LIN {X -43.0459,Y -0.6324,Z 64,A 175.5443,B 24.8515,C -2.8114,E1 24.8399,E2 -452.242} C_DIS
LIN {X -42.8004,Y -4.6329,Z 64,A 179.985,B 24.8544,C -2.7845,E1 24.8408,E2 -456.6449} C_DIS
LIN {X -42.4925,Y -6.9113,Z 64,A -176.2267,B 24.8544,C -2.7835,E1 24.8424,E2 -460.4535} C_DIS
LIN {X -41.9801,Y -9.5417,Z 64,A -173.207,B 24.8563,C -2.7664,E1 24.8441,E2 -463.45} C_DIS
LIN {X -41.3672,Y -11.9206,Z 64,A -169.4203,B 24.8566,C -2.7627,E1 24.8469,E2 -467.25} C_DIS
LIN {X -40.6957,Y -14.0446,Z 64,A -166.9986,B 24.8582,C -2.7477,E1 24.849,E2 -469.6495} C_DIS
LIN {X -40.0362,Y -15.8256,Z 64,A -163.8993,B 24.8582,C -2.7473,E1 24.8522,E2 -472.7653} C_DIS
LIN {X -38.5859,Y -19.0906,Z 64,A -159.1582,B 24.8596,C -2.734,E1 24.8578,E2 -477.5005} C_DIS
LIN {X -37.383,Y -21.3509,Z 64,A -155.9337,B 24.8608,C -2.7228,E1 24.8621,E2 -480.7152} C_DIS
LIN {X -36.011,Y -23.5919,Z 64,A -151.8552,B 24.8609,C -2.7211,E1 24.8683,E2 -484.8102} C_DIS
LIN {X -33.9335,Y -26.4939,Z 64,A -148.0687,B 24.8633,C -2.6978,E1 24.8745,E2 -488.5593} C_DIS
LIN {X -32.7195,Y -27.9783,Z 64,A -144.7571,B 24.8629,C -2.7016,E1 24.8805,E2 -491.8951} C_DIS
LIN {X -30.5092,Y -30.3738,Z 64,A -140.4648,B 24.8639,C -2.6918,E1 24.8888,E2 -496.1827} C_DIS
LIN {X -28.3095,Y -32.4332,Z 64,A -136.6606,B 24.865,C -2.6814,E1 24.8966,E2 -499.9773} C_DIS
LIN {X -26.4063,Y -34.0012,Z 64,A -132.8381,B 24.8649,C -2.6826,E1 24.905,E2 -503.8169} C_DIS
LIN {X -24.1559,Y -35.6349,Z 64,A -129.9583,B 24.8666,C -2.6658,E1 24.9115,E2 -506.6663} C_DIS
LIN {X -22.8031,Y -36.5153,Z 64,A -127.7743,B 24.8668,C -2.6631,E1 24.9167,E2 -508.8508} C_DIS
LIN {X -21.2138,Y -37.4614,Z 64,A -125.1699,B 24.867,C -2.6616,E1 24.923,E2 -511.4595} C_DIS
LIN {X -19.0637,Y -38.5993,Z 64,A -121.4922,B 24.8668,C -2.6636,E1 24.9321,E2 -515.1519} C_DIS
LIN {X -17.0057,Y -39.5497,Z 64,A -118.6789,B 24.8674,C -2.6576,E1 24.9393,E2 -517.9576} C_DIS
LIN {X -14.609,Y -40.496,Z 64,A -115.2669,B 24.8677,C -2.6543,E1 24.9482,E2 -521.3688} C_DIS
LIN {X -12.2316,Y -41.2764,Z 64,A -112.2891,B 24.8684,C -2.6469,E1 24.9561,E2 -524.3343} C_DIS
LIN {X -9.3529,Y -42.0226,Z 64,A -107.8941,B 24.868,C -2.651,E1 24.9681,E2 -528.7452} C_DIS
LIN {X -7.0809,Y -42.4642,Z 64,A -105.1078,B 24.8686,C -2.6458,E1 24.9757,E2 -531.5218} C_DIS
LIN {X -5.1708,Y -42.7388,Z 64,A -102.643,B 24.8688,C -2.6438,E1 24.9825,E2 -533.9838} C_DIS
LIN {X -3.5971,Y -42.9002,Z 64,A -100.2672,B 24.8684,C -2.6476,E1 24.9892,E2 -536.37} C_DIS
LIN {X -1.226,Y -43.0327,Z 64,A -97.3544,B 24.8687,C -2.6442,E1 24.9973,E2 -539.2753} C_DIS
LIN {X 0.3045,Y -43.0476,Z 64,A -96.1061,B 24.8698,C -2.6329,E1 25.0007,E2 -540.4966} C_DIS
Enddeposition()
LIN {X 0.3045,Y -43.0476,Z 64,A -96.1061,B 24.8698,C -2.6329,E1 25.0007,E2 -540.4966} C_DIS
Startdeposition()
$VEL.CP = VEL_PRINT
LIN {X -0.8408,Y -42.1035,Z 64,A -98.2548,B 24.8691,C -2.6404,E1 24.9947,E2 -538.3656} C_DIS
LIN {X -2.6877,Y -42.026,Z 64,A -100.418,B 24.8686,C -2.6452,E1 24.9887,E2 -536.2133} C_DIS
LIN {X -4.3067,Y -41.8908,Z 64,A -103.1544,B 24.8693,C -2.638,E1 24.9811,E2 -533.4582} C_DIS
LIN {X -7.2758,Y -41.4788,Z 64,A -106.7064,B 24.8685,C -2.6463,E1 24.9713,E2 -529.923} C_DIS
LIN {X -8.6479,Y -41.2146,Z 64,A -108.7819,B 24.8687,C -2.6447,E1 24.9656,E2 -527.8412} C_DIS
LIN {X -10.5513,Y -40.7684,Z 64,A -111.6222,B 24.8687,C -2.6436,E1 24.9579,E2 -524.9944} C_DIS
LIN {X -12.6192,Y -40.1765,Z 64,A -114.6103,B 24.8687,C -2.6448,E1 24.9499,E2 -522.0041} C_DIS
LIN {X -15.0744,Y -39.3215,Z 64,A -118.1421,B 24.8683,C -2.648,E1 24.9407,E2 -518.4726} C_DIS
LIN {X -17.3619,Y -38.3663,Z 64,A -121.5533,B 24.868,C -2.651,E1 24.9319,E2 -515.0606} C_DIS
LIN {X -19.6756,Y -37.2327,Z 64,A -124.9162,B 24.8674,C -2.6571,E1 24.9236,E2 -511.7032} C_DIS
LIN {X -21.7868,Y -36.0382,Z 64,A -128.2951,B 24.8671,C -2.6607,E1 24.9154,E2 -508.3227} C_DIS
LIN {X -23.9319,Y -34.651,Z 64,A -131.8987,B 24.8667,C -2.6645,E1 24.907,E2 -504.7162} C_DIS
LIN {X -25.7414,Y -33.3285,Z 64,A -134.4656,B 24.8656,C -2.6757,E1 24.9013,E2 -502.1668} C_DIS
LIN {X -27.559,Y -31.8423,Z 64,A -138.0378,B 24.8654,C -2.6769,E1 24.8937,E2 -498.5839} C_DIS
LIN {X -29.0326,Y -30.5047,Z 64,A -140.8361,B 24.865,C -2.6812,E1 24.888,E2 -495.7843} C_DIS
LIN {X -30.9232,Y -28.5865,Z 64,A -144.6561,B 24.8644,C -2.6871,E1 24.8806,E2 -491.9619} C_DIS
LIN {X -32.7144,Y -26.5174,Z 64,A -147.9629,B 24.8631,C -2.7004,E1 24.8747,E2 -488.6717} C_DIS
LIN {X -34.1773,Y -24.6037,Z 64,A -151.7628,B 24.8629,C -2.7021,E1 24.8683,E2 -484.8577} C_DIS
LIN {X -35.4943,Y -22.6621,Z 64,A -155.1074,B 24.8622,C -2.7084,E1 24.8632,E2 -481.5113} C_DIS
LIN {X -37.1902,Y -19.7563,Z 64,A -159.2243,B 24.8605,C -2.7256,E1 24.8576,E2 -477.414} C_DIS
Enddeposition()
END
